LIN {X 0,Y 523.889,Z 260.036,A -85,B 0,C 180,E1 -4743.726,E2 -4743.726} C_VEL
LIN {X 0,Y 523.918,Z 260.038,A -85,B 0,C 180,E1 -4746.691,E2 -4746.691} C_VEL
LIN {X 0,Y 523.956,Z 260.157,A -85,B 0,C 180,E1 -4746.98,E2 -4746.98} C_VEL
LIN {X 0,Y 524.86,Z 266.458,A -85,B 0,C 180,E1 -4748.189,E2 -4748.189} C_VEL
LIN {X 0,Y 524.6,Z 281.046,A -85,B 0,C 180,E1 -4750.841,E2 -4750.841} C_VEL
LIN {X 0,Y 524.215,Z 299.07,A -85,B 0,C 180,E1 -4754.049,E2 -4754.049} C_VEL
LIN {X 0,Y 523.903,Z 316.991,A -85,B 0,C 180,E1 -4757.214,E2 -4757.214} C_VEL
LIN {X 0,Y 523.859,Z 321.977,A -85,B 0,C 180,E1 -4758.092,E2 -4758.092} C_VEL
LIN {X 0,Y 524.896,Z 332.327,A -85,B 0,C 180,E1 -4758.281,E2 -4758.281} C_VEL
LIN {X 0,Y 524.698,Z 397.178,A -85,B 0,C 180,E1 -4759.193,E2 -4759.193} C_VEL
LIN {X 0,Y 524.555,Z 406.795,A -85,B 0,C 180,E1 -4759.41,E2 -4759.41} C_VEL
LIN {X 0,Y 524.415,Z 416.072,A -85,B 0,C 180,E1 -4759.724,E2 -4759.724} C_VEL
LIN {X 0,Y 524.265,Z 425.523,A -85,B 0,C 180,E1 -4760.16,E2 -4760.16} C_VEL
LIN {X 0,Y 524.126,Z 435.206,A -85,B 0,C 180,E1 -4760.742,E2 -4760.742} C_VEL
LIN {X 0,Y 523.895,Z 445.114,A -85,B 0,C 180,E1 -4761.516,E2 -4761.516} C_VEL
LIN {X 0,Y 523.735,Z 452.925,A -85,B 0,C 180,E1 -4762.29,E2 -4762.29} C_VEL
LIN {X 0,Y 523.66,Z 459.358,A -85,B 0,C 180,E1 -4763.064,E2 -4763.064} C_VEL
LIN {X 0,Y 523.588,Z 464.701,A -85,B 0,C 180,E1 -4763.837,E2 -4763.837} C_VEL
LIN {X 0,Y 523.484,Z 469.154,A -85,B 0,C 180,E1 -4764.609,E2 -4764.609} C_VEL
LIN {X 0,Y 523.449,Z 474.389,A -85,B 0,C 180,E1 -4765.767,E2 -4765.767} C_VEL
LIN {X 0,Y 523.406,Z 477.073,A -85,B 0,C 180,E1 -4766.537,E2 -4766.537} C_VEL
LIN {X 0,Y 523.337,Z 480.007,A -85,B 0,C 180,E1 -4767.692,E2 -4767.692} C_VEL
LIN {X 0,Y 523.274,Z 481.275,A -85,B 0,C 180,E1 -4768.462,E2 -4768.462} C_VEL
LIN {X 0,Y 523.25,Z 482.063,A -85,B 0,C 180,E1 -4769.232,E2 -4769.232} C_VEL
LIN {X 0,Y 523.251,Z 482.356,A -85,B 0,C 180,E1 -4770.001,E2 -4770.001} C_VEL
LIN {X 0,Y 523.25,Z 482.054,A -85,B 0,C 180,E1 -4770.771,E2 -4770.771} C_VEL
LIN {X 0,Y 523.274,Z 481.262,A -85,B 0,C 180,E1 -4771.541,E2 -4771.541} C_VEL
LIN {X 0,Y 523.338,Z 479.983,A -85,B 0,C 180,E1 -4772.31,E2 -4772.31} C_VEL
LIN {X 0,Y 523.407,Z 477.038,A -85,B 0,C 180,E1 -4773.465,E2 -4773.465} C_VEL
LIN {X 0,Y 523.45,Z 474.338,A -85,B 0,C 180,E1 -4774.236,E2 -4774.236} C_VEL
LIN {X 0,Y 523.484,Z 469.071,A -85,B 0,C 180,E1 -4775.394,E2 -4775.394} C_VEL
LIN {X 0,Y 523.576,Z 463.108,A -85,B 0,C 180,E1 -4776.405,E2 -4776.405} C_VEL
LIN {X 0,Y 523.705,Z 456.205,A -85,B 0,C 180,E1 -4777.326,E2 -4777.326} C_VEL
LIN {X 0,Y 523.843,Z 448.009,A -85,B 0,C 180,E1 -4778.196,E2 -4778.196} C_VEL
LIN {X 0,Y 523.981,Z 440.157,A -85,B 0,C 180,E1 -4778.874,E2 -4778.874} C_VEL
LIN {X 0,Y 524.132,Z 431.877,A -85,B 0,C 180,E1 -4779.455,E2 -4779.455} C_VEL
LIN {X 0,Y 524.28,Z 421.359,A -85,B 0,C 180,E1 -4780.037,E2 -4780.037} C_VEL
LIN {X 0,Y 524.467,Z 409.445,A -85,B 0,C 180,E1 -4780.497,E2 -4780.497} C_VEL
LIN {X 0,Y 524.616,Z 400.044,A -85,B 0,C 180,E1 -4780.738,E2 -4780.738} C_VEL
LIN {X 0,Y 524.793,Z 362.647,A -85,B 0,C 180,E1 -4781.296,E2 -4781.296} C_VEL
LIN {X 0,Y 524.773,Z 329.873,A -85,B 0,C 180,E1 -4781.752,E2 -4781.752} C_VEL
LIN {X 0,Y 523.817,Z 321.168,A -85,B 0,C 180,E1 -4781.929,E2 -4781.929} C_VEL
LIN {X 0,Y 523.987,Z 304.449,A -85,B 0,C 180,E1 -4784.765,E2 -4784.765} C_VEL
LIN {X 0,Y 524.149,Z 285.845,A -85,B 0,C 180,E1 -4787.822,E2 -4787.822} C_VEL
LIN {X 0,Y 524.255,Z 270.152,A -85,B 0,C 180,E1 -4790.4,E2 -4790.4} C_VEL
LIN {X 0,Y 524.132,Z 261.261,A -85,B 0,C 180,E1 -4791.846,E2 -4791.846} C_VEL
LIN {X 0,Y 523.953,Z 260.033,A -85,B 0,C 180,E1 -4792.061,E2 -4792.061} C_VEL
LIN {X 0,Y 523.897,Z 260.041,A -85,B 0,C 180,E1 -4794.575,E2 -4794.575} C_VEL
LIN {X 0,Y 523.92,Z 260.034,A -85,B 0,C 180,E1 -4797.704,E2 -4797.704} C_VEL
LIN {X 0,Y 523.901,Z 260.042,A -85,B 0,C 180,E1 -4800.845,E2 -4800.845} C_VEL
LIN {X 0,Y 523.863,Z 260.039,A -85,B 0,C 180,E1 -4803.717,E2 -4803.717} C_VEL
LIN {X 0,Y 523.858,Z 260.041,A -85,B 0,C 180,E1 -4806.392,E2 -4806.392} C_VEL
LIN {X 0,Y 523.903,Z 260.04,A -85,B 0,C 180,E1 -4809.087,E2 -4809.087} C_VEL
LIN {X 0,Y 523.898,Z 260.033,A -85,B 0,C 180,E1 -4812.125,E2 -4812.125} C_VEL
LIN {X 0,Y 523.944,Z 260.032,A -85,B 0,C 180,E1 -4815.311,E2 -4815.311} C_VEL
LIN {X 0,Y 523.927,Z 260.034,A -85,B 0,C 180,E1 -4818.694,E2 -4818.694} C_VEL
LIN {X 0,Y 523.922,Z 260.029,A -85,B 0,C 180,E1 -4821.896,E2 -4821.896} C_VEL
LIN {X 0,Y 523.929,Z 260.036,A -85,B 0,C 180,E1 -4824.912,E2 -4824.912} C_VEL
LIN {X 0,Y 523.949,Z 260.029,A -85,B 0,C 180,E1 -4827.679,E2 -4827.679} C_VEL
LIN {X 0,Y 523.966,Z 260.03,A -85,B 0,C 180,E1 -4830.676,E2 -4830.676} C_VEL
LIN {X 0,Y 523.941,Z 260.032,A -85,B 0,C 180,E1 -4833.724,E2 -4833.724} C_VEL
LIN {X 0,Y 523.924,Z 260.033,A -85,B 0,C 180,E1 -4836.267,E2 -4836.267} C_VEL
LIN {X 0,Y 523.958,Z 260.032,A -85,B 0,C 180,E1 -4838.764,E2 -4838.764} C_VEL
LIN {X 0,Y 523.961,Z 260.035,A -85,B 0,C 180,E1 -4841.218,E2 -4841.218} C_VEL
LIN {X 0,Y 524.175,Z 260.008,A -85,B 0,C 180,E1 -4843.643,E2 -4843.643} C_VEL
LIN {X 0,Y 524.071,Z 260.146,A -85,B 0,C 180,E1 -4844.522,E2 -4844.522} C_VEL
LIN {X 0,Y 523.648,Z 275.738,A -85,B 0,C 180,E1 -4846.808,E2 -4846.808} C_VEL
LIN {X 0,Y 523.664,Z 284.072,A -85,B 0,C 180,E1 -4848.14,E2 -4848.14} C_VEL
LIN {X 0,Y 524.911,Z 295.01,A -85,B 0,C 180,E1 -4848.33,E2 -4848.33} C_VEL
LIN {X 0,Y 524.622,Z 361.976,A -85,B 0,C 180,E1 -4849.309,E2 -4849.309} C_VEL
LIN {X 0,Y 524.525,Z 373.079,A -85,B 0,C 180,E1 -4849.6,E2 -4849.6} C_VEL
LIN {X 0,Y 524.355,Z 384.293,A -85,B 0,C 180,E1 -4850.06,E2 -4850.06} C_VEL
LIN {X 0,Y 524.207,Z 393.074,A -85,B 0,C 180,E1 -4850.544,E2 -4850.544} C_VEL
LIN {X 0,Y 524.091,Z 401.438,A -85,B 0,C 180,E1 -4851.125,E2 -4851.125} C_VEL
LIN {X 0,Y 523.938,Z 409.332,A -85,B 0,C 180,E1 -4851.803,E2 -4851.803} C_VEL
LIN {X 0,Y 523.824,Z 415.845,A -85,B 0,C 180,E1 -4852.48,E2 -4852.48} C_VEL
LIN {X 0,Y 523.672,Z 422.247,A -85,B 0,C 180,E1 -4853.281,E2 -4853.281} C_VEL
LIN {X 0,Y 523.616,Z 428.331,A -85,B 0,C 180,E1 -4854.219,E2 -4854.219} C_VEL
LIN {X 0,Y 523.471,Z 434.175,A -85,B 0,C 180,E1 -4855.376,E2 -4855.376} C_VEL
LIN {X 0,Y 523.486,Z 438.418,A -85,B 0,C 180,E1 -4856.533,E2 -4856.533} C_VEL
LIN {X 0,Y 523.339,Z 441.373,A -85,B 0,C 180,E1 -4857.687,E2 -4857.687} C_VEL
LIN {X 0,Y 523.276,Z 442.68,A -85,B 0,C 180,E1 -4858.457,E2 -4858.457} C_VEL
LIN {X 0,Y 523.255,Z 443.496,A -85,B 0,C 180,E1 -4859.227,E2 -4859.227} C_VEL
LIN {X 0,Y 523.256,Z 443.782,A -85,B 0,C 180,E1 -4859.996,E2 -4859.996} C_VEL
LIN {X 0,Y 523.256,Z 443.525,A -85,B 0,C 180,E1 -4860.766,E2 -4860.766} C_VEL
LIN {X 0,Y 523.275,Z 442.784,A -85,B 0,C 180,E1 -4861.535,E2 -4861.535} C_VEL
LIN {X 0,Y 523.34,Z 441.553,A -85,B 0,C 180,E1 -4862.305,E2 -4862.305} C_VEL
LIN {X 0,Y 523.484,Z 438.672,A -85,B 0,C 180,E1 -4863.46,E2 -4863.46} C_VEL
LIN {X 0,Y 523.455,Z 434.53,A -85,B 0,C 180,E1 -4864.616,E2 -4864.616} C_VEL
LIN {X 0,Y 523.613,Z 428.855,A -85,B 0,C 180,E1 -4865.773,E2 -4865.773} C_VEL
LIN {X 0,Y 523.666,Z 422.901,A -85,B 0,C 180,E1 -4866.713,E2 -4866.713} C_VEL
LIN {X 0,Y 523.779,Z 416.652,A -85,B 0,C 180,E1 -4867.513,E2 -4867.513} C_VEL
LIN {X 0,Y 523.983,Z 408.265,A -85,B 0,C 180,E1 -4868.383,E2 -4868.383} C_VEL
LIN {X 0,Y 524.21,Z 398.911,A -85,B 0,C 180,E1 -4869.156,E2 -4869.156} C_VEL
LIN {X 0,Y 524.363,Z 388.078,A -85,B 0,C 180,E1 -4869.835,E2 -4869.835} C_VEL
LIN {X 0,Y 524.504,Z 378.879,A -85,B 0,C 180,E1 -4870.271,E2 -4870.271} C_VEL
LIN {X 0,Y 524.587,Z 369.996,A -85,B 0,C 180,E1 -4870.586,E2 -4870.586} C_VEL
LIN {X 0,Y 524.691,Z 361.16,A -85,B 0,C 180,E1 -4870.804,E2 -4870.804} C_VEL
LIN {X 0,Y 524.859,Z 292.641,A -85,B 0,C 180,E1 -4871.798,E2 -4871.798} C_VEL
LIN {X 0,Y 523.743,Z 285.466,A -85,B 0,C 180,E1 -4871.934,E2 -4871.934} C_VEL
LIN {X 0,Y 523.895,Z 272.16,A -85,B 0,C 180,E1 -4875.01,E2 -4875.01} C_VEL
LIN {X 0,Y 524.015,Z 260.204,A -85,B 0,C 180,E1 -4877.818,E2 -4877.818} C_VEL
LIN {X 0,Y 523.939,Z 260.031,A -85,B 0,C 180,E1 -4880.406,E2 -4880.406} C_VEL
LIN {X 0,Y 523.891,Z 260.042,A -85,B 0,C 180,E1 -4882.889,E2 -4882.889} C_VEL
LIN {X 0,Y 523.88,Z 260.042,A -85,B 0,C 180,E1 -4885.417,E2 -4885.417} C_VEL
LIN {X 0,Y 523.886,Z 260.036,A -85,B 0,C 180,E1 -4887.998,E2 -4887.998} C_VEL
LIN {X 0,Y 523.884,Z 260.039,A -85,B 0,C 180,E1 -4890.87,E2 -4890.87} C_VEL
LIN {X 0,Y 523.934,Z 260.034,A -85,B 0,C 180,E1 -4893.729,E2 -4893.729} C_VEL
LIN {X 0,Y 523.906,Z 260.034,A -85,B 0,C 180,E1 -4894.216,E2 -4894.216} C_VEL
LIN {X 0,Y 523.227,Z 260.121,A -85,B 0,C 180,E1 -4894.857,E2 -4894.857} C_VEL
LIN {X 0,Y 520.334,Z 260.481,A -85,B 0,C 180,E1 -4895.897,E2 -4895.897} C_VEL
LIN {X 0,Y 517.909,Z 260.781,A -85,B 0,C 180,E1 -4896.735,E2 -4896.735} C_VEL
LIN {X 0,Y 516.892,Z 260.913,A -85,B 0,C 180,E1 -4897.383,E2 -4897.383} C_VEL
LIN {X 0,Y 516.822,Z 260.92,A -85,B 0,C 180,E1 -4897.602,E2 -4897.602} C_VEL
LIN {X 0,Y 516.849,Z 260.913,A -85,B 0,C 180,E1 -4900.405,E2 -4900.405} C_VEL
LIN {X 0,Y 516.825,Z 260.916,A -85,B 0,C 180,E1 -4902.829,E2 -4902.829} C_VEL
LIN {X 0,Y 516.86,Z 260.912,A -85,B 0,C 180,E1 -4905.002,E2 -4905.002} C_VEL
LIN {X 0,Y 516.878,Z 260.91,A -85,B 0,C 180,E1 -4908.394,E2 -4908.394} C_VEL
LIN {X 0,Y 516.839,Z 260.916,A -85,B 0,C 180,E1 -4911.279,E2 -4911.279} C_VEL
LIN {X 0,Y 516.845,Z 260.918,A -85,B 0,C 180,E1 -4914.217,E2 -4914.217} C_VEL
LIN {X 0,Y 516.85,Z 260.912,A -85,B 0,C 180,E1 -4917.049,E2 -4917.049} C_VEL
LIN {X 0,Y 516.852,Z 260.918,A -85,B 0,C 180,E1 -4919.793,E2 -4919.793} C_VEL
LIN {X 0,Y 516.88,Z 260.914,A -85,B 0,C 180,E1 -4922.464,E2 -4922.464} C_VEL
LIN {X 0,Y 516.865,Z 260.911,A -85,B 0,C 180,E1 -4925.068,E2 -4925.068} C_VEL
LIN {X 0,Y 516.832,Z 260.921,A -85,B 0,C 180,E1 -4928.459,E2 -4928.459} C_VEL
LIN {X 0,Y 516.849,Z 260.914,A -85,B 0,C 180,E1 -4930.952,E2 -4930.952} C_VEL
LIN {X 0,Y 516.857,Z 260.912,A -85,B 0,C 180,E1 -4933.407,E2 -4933.407} C_VEL
LIN {X 0,Y 516.839,Z 260.915,A -85,B 0,C 180,E1 -4935.831,E2 -4935.831} C_VEL
LIN {X 0,Y 516.946,Z 260.905,A -85,B 0,C 180,E1 -4938.232,E2 -4938.232} C_VEL
LIN {X 0,Y 516.916,Z 260.905,A -85,B 0,C 180,E1 -4941.398,E2 -4941.398} C_VEL
LIN {X 0,Y 517.005,Z 260.9,A -85,B 0,C 180,E1 -4944.538,E2 -4944.538} C_VEL
LIN {X 0,Y 517.022,Z 260.891,A -85,B 0,C 180,E1 -4947.662,E2 -4947.662} C_VEL
LIN {X 0,Y 517.039,Z 260.895,A -85,B 0,C 180,E1 -4950.778,E2 -4950.778} C_VEL
LIN {X 0,Y 516.988,Z 260.901,A -85,B 0,C 180,E1 -4953.116,E2 -4953.116} C_VEL
LIN {X 0,Y 516.949,Z 260.9,A -85,B 0,C 180,E1 -4956.242,E2 -4956.242} C_VEL
LIN {X 0,Y 516.905,Z 260.911,A -85,B 0,C 180,E1 -4959.389,E2 -4959.389} C_VEL
LIN {X 0,Y 516.92,Z 260.905,A -85,B 0,C 180,E1 -4961.824,E2 -4961.824} C_VEL
LIN {X 0,Y 516.88,Z 260.915,A -85,B 0,C 180,E1 -4965.147,E2 -4965.147} C_VEL
LIN {X 0,Y 516.864,Z 260.911,A -85,B 0,C 180,E1 -4968.223,E2 -4968.223} C_VEL
LIN {X 0,Y 516.853,Z 260.913,A -85,B 0,C 180,E1 -4970.702,E2 -4970.702} C_VEL
LIN {X 0,Y 516.817,Z 260.922,A -85,B 0,C 180,E1 -4973.224,E2 -4973.224} C_VEL
LIN {X 0,Y 516.889,Z 260.909,A -85,B 0,C 180,E1 -4976.199,E2 -4976.199} C_VEL
LIN {X 0,Y 516.876,Z 260.913,A -85,B 0,C 180,E1 -4979.305,E2 -4979.305} C_VEL
LIN {X 0,Y 516.843,Z 260.914,A -85,B 0,C 180,E1 -4982.546,E2 -4982.546} C_VEL
LIN {X 0,Y 516.827,Z 260.918,A -85,B 0,C 180,E1 -4985.335,E2 -4985.335} C_VEL
LIN {X 0,Y 516.828,Z 260.921,A -85,B 0,C 180,E1 -4987.946,E2 -4987.946} C_VEL
LIN {X 0,Y 516.866,Z 260.911,A -85,B 0,C 180,E1 -4990.741,E2 -4990.741} C_VEL
LIN {X 0,Y 516.831,Z 260.922,A -85,B 0,C 180,E1 -4993.906,E2 -4993.906} C_VEL
LIN {X 0,Y 516.832,Z 260.921,A -85,B 0,C 180,E1 -4996.11,E2 -4996.11} C_VEL
LIN {X 0,Y 516.856,Z 260.912,A -85,B 0,C 180,E1 -4999.264,E2 -4999.264} C_VEL
LIN {X 0,Y 516.819,Z 260.923,A -85,B 0,C 180,E1 -5002.278,E2 -5002.278} C_VEL
LIN {X 0,Y 516.853,Z 260.913,A -85,B 0,C 180,E1 -5005.18,E2 -5005.18} C_VEL
LIN {X 0,Y 516.835,Z 260.917,A -85,B 0,C 180,E1 -5007.979,E2 -5007.979} C_VEL
LIN {X 0,Y 516.88,Z 260.915,A -85,B 0,C 180,E1 -5010.699,E2 -5010.699} C_VEL
LIN {X 0,Y 516.875,Z 260.91,A -85,B 0,C 180,E1 -5013.815,E2 -5013.815} C_VEL
LIN {X 0,Y 516.823,Z 260.922,A -85,B 0,C 180,E1 -5016.78,E2 -5016.78} C_VEL
LIN {X 0,Y 516.904,Z 260.906,A -85,B 0,C 180,E1 -5019.737,E2 -5019.737} C_VEL
LIN {X 0,Y 516.867,Z 260.916,A -85,B 0,C 180,E1 -5022.599,E2 -5022.599} C_VEL
LIN {X 0,Y 516.911,Z 260.911,A -85,B 0,C 180,E1 -5025.034,E2 -5025.034} C_VEL
LIN {X 0,Y 516.94,Z 260.902,A -85,B 0,C 180,E1 -5028.238,E2 -5028.238} C_VEL
LIN {X 0,Y 516.927,Z 260.908,A -85,B 0,C 180,E1 -5031.403,E2 -5031.403} C_VEL
LIN {X 0,Y 516.962,Z 260.9,A -85,B 0,C 180,E1 -5033.761,E2 -5033.761} C_VEL
LIN {X 0,Y 516.954,Z 260.904,A -85,B 0,C 180,E1 -5036.887,E2 -5036.887} C_VEL
LIN {X 0,Y 517.075,Z 260.891,A -85,B 0,C 180,E1 -5039.225,E2 -5039.225} C_VEL
LIN {X 0,Y 517.056,Z 260.887,A -85,B 0,C 180,E1 -5042.341,E2 -5042.341} C_VEL
LIN {X 0,Y 516.995,Z 260.901,A -85,B 0,C 180,E1 -5045.464,E2 -5045.464} C_VEL
LIN {X 0,Y 516.938,Z 260.901,A -85,B 0,C 180,E1 -5048.604,E2 -5048.604} C_VEL
LIN {X 0,Y 516.94,Z 260.907,A -85,B 0,C 180,E1 -5051.81,E2 -5051.81} C_VEL
LIN {X 0,Y 516.932,Z 260.904,A -85,B 0,C 180,E1 -5055.149,E2 -5055.149} C_VEL
LIN {X 0,Y 516.867,Z 260.914,A -85,B 0,C 180,E1 -5058.227,E2 -5058.227} C_VEL
LIN {X 0,Y 516.89,Z 260.908,A -85,B 0,C 180,E1 -5060.705,E2 -5060.705} C_VEL
LIN {X 0,Y 516.848,Z 260.913,A -85,B 0,C 180,E1 -5063.227,E2 -5063.227} C_VEL
LIN {X 0,Y 516.872,Z 260.915,A -85,B 0,C 180,E1 -5066.185,E2 -5066.185} C_VEL
LIN {X 0,Y 516.914,Z 260.905,A -85,B 0,C 180,E1 -5069.308,E2 -5069.308} C_VEL
LIN {X 0,Y 516.888,Z 260.912,A -85,B 0,C 180,E1 -5072.546,E2 -5072.546} C_VEL
LIN {X 0,Y 516.848,Z 260.913,A -85,B 0,C 180,E1 -5075.33,E2 -5075.33} C_VEL
LIN {X 0,Y 516.866,Z 260.915,A -85,B 0,C 180,E1 -5078.72,E2 -5078.72} C_VEL
LIN {X 0,Y 516.849,Z 260.914,A -85,B 0,C 180,E1 -5081.784,E2 -5081.784} C_VEL
LIN {X 0,Y 516.893,Z 260.91,A -85,B 0,C 180,E1 -5085.009,E2 -5085.009} C_VEL
LIN {X 0,Y 516.852,Z 260.918,A -85,B 0,C 180,E1 -5088.409,E2 -5088.409} C_VEL
LIN {X 0,Y 516.873,Z 260.911,A -85,B 0,C 180,E1 -5091.286,E2 -5091.286} C_VEL
LIN {X 0,Y 516.854,Z 260.914,A -85,B 0,C 180,E1 -5094.221,E2 -5094.221} C_VEL
LIN {X 0,Y 516.878,Z 260.915,A -85,B 0,C 180,E1 -5097.054,E2 -5097.054} C_VEL
LIN {X 0,Y 516.85,Z 260.913,A -85,B 0,C 180,E1 -5099.796,E2 -5099.796} C_VEL
LIN {X 0,Y 516.868,Z 260.912,A -85,B 0,C 180,E1 -5102.466,E2 -5102.466} C_VEL
LIN {X 0,Y 516.87,Z 260.915,A -85,B 0,C 180,E1 -5105.648,E2 -5105.648} C_VEL
LIN {X 0,Y 516.903,Z 260.981,A -85,B 0,C 180,E1 -5106.832,E2 -5106.832} C_VEL
LIN {X 0,Y 517.891,Z 267.442,A -85,B 0,C 180,E1 -5108.089,E2 -5108.089} C_VEL
LIN {X 0,Y 517.585,Z 281.977,A -85,B 0,C 180,E1 -5110.777,E2 -5110.777} C_VEL
LIN {X 0,Y 517.177,Z 298.875,A -85,B 0,C 180,E1 -5113.826,E2 -5113.826} C_VEL
LIN {X 0,Y 516.885,Z 315.646,A -85,B 0,C 180,E1 -5116.837,E2 -5116.837} C_VEL
LIN {X 0,Y 516.816,Z 321.814,A -85,B 0,C 180,E1 -5117.939,E2 -5117.939} C_VEL
LIN {X 0,Y 517.959,Z 331.933,A -85,B 0,C 180,E1 -5118.121,E2 -5118.121} C_VEL
LIN {X 0,Y 517.695,Z 397.549,A -85,B 0,C 180,E1 -5119.07,E2 -5119.07} C_VEL
LIN {X 0,Y 517.537,Z 407.745,A -85,B 0,C 180,E1 -5119.314,E2 -5119.314} C_VEL
LIN {X 0,Y 517.367,Z 417.888,A -85,B 0,C 180,E1 -5119.682,E2 -5119.682} C_VEL
LIN {X 0,Y 517.166,Z 428.671,A -85,B 0,C 180,E1 -5120.221,E2 -5120.221} C_VEL
LIN {X 0,Y 516.991,Z 438.738,A -85,B 0,C 180,E1 -5120.909,E2 -5120.909} C_VEL
LIN {X 0,Y 516.813,Z 446.774,A -85,B 0,C 180,E1 -5121.595,E2 -5121.595} C_VEL
LIN {X 0,Y 516.692,Z 452.559,A -85,B 0,C 180,E1 -5122.184,E2 -5122.184} C_VEL
LIN {X 0,Y 516.593,Z 459.014,A -85,B 0,C 180,E1 -5122.968,E2 -5122.968} C_VEL
LIN {X 0,Y 516.495,Z 464.377,A -85,B 0,C 180,E1 -5123.752,E2 -5123.752} C_VEL
LIN {X 0,Y 516.421,Z 468.849,A -85,B 0,C 180,E1 -5124.535,E2 -5124.535} C_VEL
LIN {X 0,Y 516.34,Z 474.1,A -85,B 0,C 180,E1 -5125.708,E2 -5125.708} C_VEL
LIN {X 0,Y 516.324,Z 476.795,A -85,B 0,C 180,E1 -5126.49,E2 -5126.49} C_VEL
LIN {X 0,Y 516.264,Z 479.741,A -85,B 0,C 180,E1 -5127.661,E2 -5127.661} C_VEL
LIN {X 0,Y 516.192,Z 481.013,A -85,B 0,C 180,E1 -5128.441,E2 -5128.441} C_VEL
LIN {X 0,Y 516.16,Z 481.804,A -85,B 0,C 180,E1 -5129.221,E2 -5129.221} C_VEL
LIN {X 0,Y 516.158,Z 482.095,A -85,B 0,C 180,E1 -5130.001,E2 -5130.001} C_VEL
LIN {X 0,Y 516.16,Z 481.79,A -85,B 0,C 180,E1 -5130.781,E2 -5130.781} C_VEL
LIN {X 0,Y 516.192,Z 480.994,A -85,B 0,C 180,E1 -5131.562,E2 -5131.562} C_VEL
LIN {X 0,Y 516.264,Z 479.708,A -85,B 0,C 180,E1 -5132.342,E2 -5132.342} C_VEL
LIN {X 0,Y 516.325,Z 476.742,A -85,B 0,C 180,E1 -5133.513,E2 -5133.513} C_VEL
LIN {X 0,Y 516.341,Z 474.032,A -85,B 0,C 180,E1 -5134.295,E2 -5134.295} C_VEL
LIN {X 0,Y 516.422,Z 468.734,A -85,B 0,C 180,E1 -5135.468,E2 -5135.468} C_VEL
LIN {X 0,Y 516.508,Z 461.774,A -85,B 0,C 180,E1 -5136.634,E2 -5136.634} C_VEL
LIN {X 0,Y 516.628,Z 455.794,A -85,B 0,C 180,E1 -5137.427,E2 -5137.427} C_VEL
LIN {X 0,Y 516.761,Z 447.559,A -85,B 0,C 180,E1 -5138.31,E2 -5138.31} C_VEL
LIN {X 0,Y 516.945,Z 439.657,A -85,B 0,C 180,E1 -5138.996,E2 -5138.996} C_VEL
LIN {X 0,Y 517.083,Z 431.321,A -85,B 0,C 180,E1 -5139.585,E2 -5139.585} C_VEL
LIN {X 0,Y 517.284,Z 420.731,A -85,B 0,C 180,E1 -5140.174,E2 -5140.174} C_VEL
LIN {X 0,Y 517.463,Z 409.407,A -85,B 0,C 180,E1 -5140.616,E2 -5140.616} C_VEL
LIN {X 0,Y 517.618,Z 400.166,A -85,B 0,C 180,E1 -5140.86,E2 -5140.86} C_VEL
LIN {X 0,Y 517.778,Z 370.892,A -85,B 0,C 180,E1 -5141.313,E2 -5141.313} C_VEL
LIN {X 0,Y 517.811,Z 330.227,A -85,B 0,C 180,E1 -5141.902,E2 -5141.902} C_VEL
LIN {X 0,Y 516.737,Z 320.994,A -85,B 0,C 180,E1 -5142.071,E2 -5142.071} C_VEL
LIN {X 0,Y 516.909,Z 302.864,A -85,B 0,C 180,E1 -5145.128,E2 -5145.128} C_VEL
LIN {X 0,Y 517.047,Z 287.661,A -85,B 0,C 180,E1 -5147.669,E2 -5147.669} C_VEL
LIN {X 0,Y 517.201,Z 272.926,A -85,B 0,C 180,E1 -5150.104,E2 -5150.104} C_VEL
LIN {X 0,Y 517.192,Z 262.999,A -85,B 0,C 180,E1 -5151.735,E2 -5151.735} C_VEL
LIN {X 0,Y 516.906,Z 260.911,A -85,B 0,C 180,E1 -5152.115,E2 -5152.115} C_VEL
LIN {X 0,Y 516.833,Z 260.923,A -85,B 0,C 180,E1 -5154.933,E2 -5154.933} C_VEL
LIN {X 0,Y 516.864,Z 260.913,A -85,B 0,C 180,E1 -5157.89,E2 -5157.89} C_VEL
LIN {X 0,Y 516.854,Z 260.918,A -85,B 0,C 180,E1 -5161.113,E2 -5161.113} C_VEL
LIN {X 0,Y 516.829,Z 260.915,A -85,B 0,C 180,E1 -5163.951,E2 -5163.951} C_VEL
LIN {X 0,Y 516.803,Z 260.924,A -85,B 0,C 180,E1 -5166.753,E2 -5166.753} C_VEL
LIN {X 0,Y 516.838,Z 260.913,A -85,B 0,C 180,E1 -5169.726,E2 -5169.726} C_VEL
LIN {X 0,Y 516.849,Z 260.919,A -85,B 0,C 180,E1 -5172.836,E2 -5172.836} C_VEL
LIN {X 0,Y 516.91,Z 260.912,A -85,B 0,C 180,E1 -5175.006,E2 -5175.006} C_VEL
LIN {X 0,Y 516.863,Z 260.91,A -85,B 0,C 180,E1 -5178.406,E2 -5178.406} C_VEL
LIN {X 0,Y 516.886,Z 260.911,A -85,B 0,C 180,E1 -5181.282,E2 -5181.282} C_VEL
LIN {X 0,Y 516.87,Z 260.909,A -85,B 0,C 180,E1 -5184.217,E2 -5184.217} C_VEL
LIN {X 0,Y 516.895,Z 260.914,A -85,B 0,C 180,E1 -5187.05,E2 -5187.05} C_VEL
LIN {X 0,Y 516.884,Z 260.909,A -85,B 0,C 180,E1 -5189.793,E2 -5189.793} C_VEL
LIN {X 0,Y 516.893,Z 260.909,A -85,B 0,C 180,E1 -5192.463,E2 -5192.463} C_VEL
LIN {X 0,Y 516.873,Z 260.919,A -85,B 0,C 180,E1 -5195.067,E2 -5195.067} C_VEL
LIN {X 0,Y 516.883,Z 260.913,A -85,B 0,C 180,E1 -5197.619,E2 -5197.619} C_VEL
LIN {X 0,Y 516.944,Z 260.901,A -85,B 0,C 180,E1 -5200.127,E2 -5200.127} C_VEL
LIN {X 0,Y 517.085,Z 260.892,A -85,B 0,C 180,E1 -5203.413,E2 -5203.413} C_VEL
LIN {X 0,Y 516.978,Z 261.072,A -85,B 0,C 180,E1 -5204.565,E2 -5204.565} C_VEL
LIN {X 0,Y 516.589,Z 276.65,A -85,B 0,C 180,E1 -5206.825,E2 -5206.825} C_VEL
LIN {X 0,Y 516.632,Z 284.166,A -85,B 0,C 180,E1 -5207.976,E2 -5207.976} C_VEL
LIN {X 0,Y 517.975,Z 295.466,A -85,B 0,C 180,E1 -5208.178,E2 -5208.178} C_VEL
LIN {X 0,Y 517.648,Z 362.688,A -85,B 0,C 180,E1 -5209.188,E2 -5209.188} C_VEL
LIN {X 0,Y 517.533,Z 373.605,A -85,B 0,C 180,E1 -5209.482,E2 -5209.482} C_VEL
LIN {X 0,Y 517.354,Z 384.247,A -85,B 0,C 180,E1 -5209.924,E2 -5209.924} C_VEL
LIN {X 0,Y 517.2,Z 393.084,A -85,B 0,C 180,E1 -5210.415,E2 -5210.415} C_VEL
LIN {X 0,Y 517.087,Z 401.494,A -85,B 0,C 180,E1 -5211.004,E2 -5211.004} C_VEL
LIN {X 0,Y 516.923,Z 409.433,A -85,B 0,C 180,E1 -5211.691,E2 -5211.691} C_VEL
LIN {X 0,Y 516.782,Z 415.979,A -85,B 0,C 180,E1 -5212.377,E2 -5212.377} C_VEL
LIN {X 0,Y 516.628,Z 421.824,A -85,B 0,C 180,E1 -5213.11,E2 -5213.11} C_VEL
LIN {X 0,Y 516.628,Z 427.34,A -85,B 0,C 180,E1 -5213.945,E2 -5213.945} C_VEL
LIN {X 0,Y 516.399,Z 432.588,A -85,B 0,C 180,E1 -5214.921,E2 -5214.921} C_VEL
LIN {X 0,Y 516.387,Z 437.439,A -85,B 0,C 180,E1 -5216.094,E2 -5216.094} C_VEL
LIN {X 0,Y 516.375,Z 439.806,A -85,B 0,C 180,E1 -5216.875,E2 -5216.875} C_VEL
LIN {X 0,Y 516.269,Z 441.617,A -85,B 0,C 180,E1 -5217.656,E2 -5217.656} C_VEL
LIN {X 0,Y 516.193,Z 442.925,A -85,B 0,C 180,E1 -5218.436,E2 -5218.436} C_VEL
LIN {X 0,Y 516.165,Z 443.747,A -85,B 0,C 180,E1 -5219.216,E2 -5219.216} C_VEL
LIN {X 0,Y 516.163,Z 444.044,A -85,B 0,C 180,E1 -5219.996,E2 -5219.996} C_VEL
LIN {X 0,Y 516.166,Z 443.772,A -85,B 0,C 180,E1 -5220.776,E2 -5220.776} C_VEL
LIN {X 0,Y 516.192,Z 443.021,A -85,B 0,C 180,E1 -5221.556,E2 -5221.556} C_VEL
LIN {X 0,Y 516.269,Z 441.784,A -85,B 0,C 180,E1 -5222.337,E2 -5222.337} C_VEL
LIN {X 0,Y 516.389,Z 438.889,A -85,B 0,C 180,E1 -5223.507,E2 -5223.507} C_VEL
LIN {X 0,Y 516.366,Z 434.728,A -85,B 0,C 180,E1 -5224.68,E2 -5224.68} C_VEL
LIN {X 0,Y 516.57,Z 429.033,A -85,B 0,C 180,E1 -5225.852,E2 -5225.852} C_VEL
LIN {X 0,Y 516.616,Z 423.523,A -85,B 0,C 180,E1 -5226.737,E2 -5226.737} C_VEL
LIN {X 0,Y 516.74,Z 416.759,A -85,B 0,C 180,E1 -5227.616,E2 -5227.616} C_VEL
LIN {X 0,Y 516.918,Z 409.364,A -85,B 0,C 180,E1 -5228.4,E2 -5228.4} C_VEL
LIN {X 0,Y 517.114,Z 401.449,A -85,B 0,C 180,E1 -5229.086,E2 -5229.086} C_VEL
LIN {X 0,Y 517.303,Z 391.56,A -85,B 0,C 180,E1 -5229.773,E2 -5229.773} C_VEL
LIN {X 0,Y 517.487,Z 381.153,A -85,B 0,C 180,E1 -5230.313,E2 -5230.313} C_VEL
LIN {X 0,Y 517.604,Z 370.556,A -85,B 0,C 180,E1 -5230.706,E2 -5230.706} C_VEL
LIN {X 0,Y 517.688,Z 361.917,A -85,B 0,C 180,E1 -5230.927,E2 -5230.927} C_VEL
LIN {X 0,Y 517.821,Z 292.671,A -85,B 0,C 180,E1 -5231.961,E2 -5231.961} C_VEL
LIN {X 0,Y 516.713,Z 285.633,A -85,B 0,C 180,E1 -5232.099,E2 -5232.099} C_VEL
LIN {X 0,Y 516.859,Z 272.721,A -85,B 0,C 180,E1 -5235.109,E2 -5235.109} C_VEL
LIN {X 0,Y 517.04,Z 262.042,A -85,B 0,C 180,E1 -5237.641,E2 -5237.641} C_VEL
LIN {X 0,Y 516.929,Z 260.907,A -85,B 0,C 180,E1 -5237.946,E2 -5237.946} C_VEL
LIN {X 0,Y 516.888,Z 260.912,A -85,B 0,C 180,E1 -5240.697,E2 -5240.697} C_VEL
LIN {X 0,Y 516.841,Z 260.92,A -85,B 0,C 180,E1 -5243.219,E2 -5243.219} C_VEL
LIN {X 0,Y 516.863,Z 260.911,A -85,B 0,C 180,E1 -5246.177,E2 -5246.177} C_VEL
LIN {X 0,Y 516.882,Z 260.914,A -85,B 0,C 180,E1 -5249.301,E2 -5249.301} C_VEL
LIN {X 0,Y 516.87,Z 260.91,A -85,B 0,C 180,E1 -5252.538,E2 -5252.538} C_VEL
LIN {X 0,Y 516.837,Z 260.92,A -85,B 0,C 180,E1 -5255.324,E2 -5255.324} C_VEL
LIN {X 0,Y 516.822,Z 260.92,A -85,B 0,C 180,E1 -5257.602,E2 -5257.602} C_VEL
LIN {X 0,Y 516.188,Z 261.004,A -85,B 0,C 180,E1 -5258.252,E2 -5258.252} C_VEL
LIN {X 0,Y 513.335,Z 261.357,A -85,B 0,C 180,E1 -5259.308,E2 -5259.308} C_VEL
LIN {X 0,Y 510.908,Z 261.654,A -85,B 0,C 180,E1 -5260.158,E2 -5260.158} C_VEL
LIN {X 0,Y 509.874,Z 261.782,A -85,B 0,C 180,E1 -5260.814,E2 -5260.814} C_VEL
LIN {X 0,Y 509.795,Z 261.793,A -85,B 0,C 180,E1 -5261.037,E2 -5261.037} C_VEL
LIN {X 0,Y 509.787,Z 261.795,A -85,B 0,C 180,E1 -5264.202,E2 -5264.202} C_VEL
LIN {X 0,Y 509.786,Z 261.793,A -85,B 0,C 180,E1 -5266.933,E2 -5266.933} C_VEL
LIN {X 0,Y 509.799,Z 261.797,A -85,B 0,C 180,E1 -5269.613,E2 -5269.613} C_VEL
LIN {X 0,Y 509.777,Z 261.794,A -85,B 0,C 180,E1 -5272.655,E2 -5272.655} C_VEL
LIN {X 0,Y 509.815,Z 261.795,A -85,B 0,C 180,E1 -5275.793,E2 -5275.793} C_VEL
LIN {X 0,Y 509.8,Z 261.792,A -85,B 0,C 180,E1 -5278.716,E2 -5278.716} C_VEL
LIN {X 0,Y 509.849,Z 261.791,A -85,B 0,C 180,E1 -5281.895,E2 -5281.895} C_VEL
LIN {X 0,Y 509.831,Z 261.79,A -85,B 0,C 180,E1 -5284.7,E2 -5284.7} C_VEL
LIN {X 0,Y 509.775,Z 261.794,A -85,B 0,C 180,E1 -5287.454,E2 -5287.454} C_VEL
LIN {X 0,Y 509.862,Z 261.786,A -85,B 0,C 180,E1 -5289.841,E2 -5289.841} C_VEL
LIN {X 0,Y 509.828,Z 261.788,A -85,B 0,C 180,E1 -5293.172,E2 -5293.172} C_VEL
LIN {X 0,Y 509.807,Z 261.79,A -85,B 0,C 180,E1 -5295.631,E2 -5295.631} C_VEL
LIN {X 0,Y 509.872,Z 261.787,A -85,B 0,C 180,E1 -5298.872,E2 -5298.872} C_VEL
LIN {X 0,Y 509.893,Z 261.781,A -85,B 0,C 180,E1 -5302.076,E2 -5302.076} C_VEL
LIN {X 0,Y 509.951,Z 261.777,A -85,B 0,C 180,E1 -5304.463,E2 -5304.463} C_VEL
LIN {X 0,Y 509.995,Z 261.767,A -85,B 0,C 180,E1 -5307.629,E2 -5307.629} C_VEL
LIN {X 0,Y 509.99,Z 261.767,A -85,B 0,C 180,E1 -5309.999,E2 -5309.999} C_VEL
LIN {X 0,Y 509.929,Z 261.78,A -85,B 0,C 180,E1 -5313.159,E2 -5313.159} C_VEL
LIN {X 0,Y 509.917,Z 261.777,A -85,B 0,C 180,E1 -5316.329,E2 -5316.329} C_VEL
LIN {X 0,Y 509.889,Z 261.783,A -85,B 0,C 180,E1 -5318.719,E2 -5318.719} C_VEL
LIN {X 0,Y 509.888,Z 261.781,A -85,B 0,C 180,E1 -5321.93,E2 -5321.93} C_VEL
LIN {X 0,Y 509.83,Z 261.793,A -85,B 0,C 180,E1 -5325.242,E2 -5325.242} C_VEL
LIN {X 0,Y 509.826,Z 261.789,A -85,B 0,C 180,E1 -5328.002,E2 -5328.002} C_VEL
LIN {X 0,Y 509.792,Z 261.795,A -85,B 0,C 180,E1 -5331.002,E2 -5331.002} C_VEL
LIN {X 0,Y 509.782,Z 261.799,A -85,B 0,C 180,E1 -5333.564,E2 -5333.564} C_VEL
LIN {X 0,Y 509.857,Z 261.784,A -85,B 0,C 180,E1 -5336.381,E2 -5336.381} C_VEL
LIN {X 0,Y 509.826,Z 261.788,A -85,B 0,C 180,E1 -5338.845,E2 -5338.845} C_VEL
LIN {X 0,Y 509.769,Z 261.801,A -85,B 0,C 180,E1 -5341.592,E2 -5341.592} C_VEL
LIN {X 0,Y 509.798,Z 261.793,A -85,B 0,C 180,E1 -5344.415,E2 -5344.415} C_VEL
LIN {X 0,Y 509.764,Z 261.797,A -85,B 0,C 180,E1 -5347.343,E2 -5347.343} C_VEL
LIN {X 0,Y 509.83,Z 261.791,A -85,B 0,C 180,E1 -5350.381,E2 -5350.381} C_VEL
LIN {X 0,Y 509.789,Z 261.792,A -85,B 0,C 180,E1 -5353.067,E2 -5353.067} C_VEL
LIN {X 0,Y 509.78,Z 261.798,A -85,B 0,C 180,E1 -5355.795,E2 -5355.795} C_VEL
LIN {X 0,Y 509.817,Z 261.793,A -85,B 0,C 180,E1 -5358.579,E2 -5358.579} C_VEL
LIN {X 0,Y 509.806,Z 261.793,A -85,B 0,C 180,E1 -5361.79,E2 -5361.79} C_VEL
LIN {X 0,Y 509.803,Z 261.796,A -85,B 0,C 180,E1 -5364.627,E2 -5364.627} C_VEL
LIN {X 0,Y 509.822,Z 261.788,A -85,B 0,C 180,E1 -5367.485,E2 -5367.485} C_VEL
LIN {X 0,Y 509.818,Z 261.794,A -85,B 0,C 180,E1 -5370.278,E2 -5370.278} C_VEL
LIN {X 0,Y 509.839,Z 261.79,A -85,B 0,C 180,E1 -5372.948,E2 -5372.948} C_VEL
LIN {X 0,Y 509.806,Z 261.79,A -85,B 0,C 180,E1 -5375.577,E2 -5375.577} C_VEL
LIN {X 0,Y 509.787,Z 261.794,A -85,B 0,C 180,E1 -5378.153,E2 -5378.153} C_VEL
LIN {X 0,Y 509.825,Z 261.794,A -85,B 0,C 180,E1 -5380.685,E2 -5380.685} C_VEL
LIN {X 0,Y 509.839,Z 261.791,A -85,B 0,C 180,E1 -5383.178,E2 -5383.178} C_VEL
LIN {X 0,Y 509.828,Z 261.788,A -85,B 0,C 180,E1 -5385.638,E2 -5385.638} C_VEL
LIN {X 0,Y 509.884,Z 261.787,A -85,B 0,C 180,E1 -5388.879,E2 -5388.879} C_VEL
LIN {X 0,Y 509.896,Z 261.779,A -85,B 0,C 180,E1 -5392.082,E2 -5392.082} C_VEL
LIN {X 0,Y 509.946,Z 261.774,A -85,B 0,C 180,E1 -5394.468,E2 -5394.468} C_VEL
LIN {X 0,Y 510.025,Z 261.767,A -85,B 0,C 180,E1 -5397.635,E2 -5397.635} C_VEL
LIN {X 0,Y 510.014,Z 261.765,A -85,B 0,C 180,E1 -5400.004,E2 -5400.004} C_VEL
LIN {X 0,Y 510.027,Z 261.763,A -85,B 0,C 180,E1 -5402.373,E2 -5402.373} C_VEL
LIN {X 0,Y 509.946,Z 261.778,A -85,B 0,C 180,E1 -5405.54,E2 -5405.54} C_VEL
LIN {X 0,Y 509.887,Z 261.78,A -85,B 0,C 180,E1 -5408.724,E2 -5408.724} C_VEL
LIN {X 0,Y 509.892,Z 261.784,A -85,B 0,C 180,E1 -5411.935,E2 -5411.935} C_VEL
LIN {X 0,Y 509.884,Z 261.783,A -85,B 0,C 180,E1 -5415.245,E2 -5415.245} C_VEL
LIN {X 0,Y 509.827,Z 261.789,A -85,B 0,C 180,E1 -5418.488,E2 -5418.488} C_VEL
LIN {X 0,Y 509.833,Z 261.787,A -85,B 0,C 180,E1 -5421.005,E2 -5421.005} C_VEL
LIN {X 0,Y 509.81,Z 261.793,A -85,B 0,C 180,E1 -5423.567,E2 -5423.567} C_VEL
LIN {X 0,Y 509.808,Z 261.794,A -85,B 0,C 180,E1 -5426.36,E2 -5426.36} C_VEL
LIN {X 0,Y 509.843,Z 261.786,A -85,B 0,C 180,E1 -5428.849,E2 -5428.849} C_VEL
LIN {X 0,Y 509.813,Z 261.791,A -85,B 0,C 180,E1 -5431.593,E2 -5431.593} C_VEL
LIN {X 0,Y 509.828,Z 261.793,A -85,B 0,C 180,E1 -5434.418,E2 -5434.418} C_VEL
LIN {X 0,Y 509.787,Z 261.792,A -85,B 0,C 180,E1 -5437.346,E2 -5437.346} C_VEL
LIN {X 0,Y 509.809,Z 261.795,A -85,B 0,C 180,E1 -5440.387,E2 -5440.387} C_VEL
LIN {X 0,Y 509.803,Z 261.79,A -85,B 0,C 180,E1 -5443.576,E2 -5443.576} C_VEL
LIN {X 0,Y 509.79,Z 261.799,A -85,B 0,C 180,E1 -5446.428,E2 -5446.428} C_VEL
LIN {X 0,Y 509.812,Z 261.789,A -85,B 0,C 180,E1 -5449.618,E2 -5449.618} C_VEL
LIN {X 0,Y 509.804,Z 261.797,A -85,B 0,C 180,E1 -5452.66,E2 -5452.66} C_VEL
LIN {X 0,Y 509.837,Z 261.786,A -85,B 0,C 180,E1 -5455.803,E2 -5455.803} C_VEL
LIN {X 0,Y 509.837,Z 261.793,A -85,B 0,C 180,E1 -5458.724,E2 -5458.724} C_VEL
LIN {X 0,Y 509.834,Z 261.792,A -85,B 0,C 180,E1 -5461.155,E2 -5461.155} C_VEL
LIN {X 0,Y 509.836,Z 261.787,A -85,B 0,C 180,E1 -5463.827,E2 -5463.827} C_VEL
LIN {X 0,Y 509.862,Z 261.934,A -85,B 0,C 180,E1 -5466.709,E2 -5466.709} C_VEL
LIN {X 0,Y 510.885,Z 268.395,A -85,B 0,C 180,E1 -5467.986,E2 -5467.986} C_VEL
LIN {X 0,Y 510.636,Z 281.817,A -85,B 0,C 180,E1 -5470.505,E2 -5470.505} C_VEL
LIN {X 0,Y 510.184,Z 298.655,A -85,B 0,C 180,E1 -5473.598,E2 -5473.598} C_VEL
LIN {X 0,Y 509.851,Z 315.417,A -85,B 0,C 180,E1 -5476.652,E2 -5476.652} C_VEL
LIN {X 0,Y 509.744,Z 321.538,A -85,B 0,C 180,E1 -5477.76,E2 -5477.76} C_VEL
LIN {X 0,Y 511.011,Z 333.503,A -85,B 0,C 180,E1 -5477.985,E2 -5477.985} C_VEL
LIN {X 0,Y 510.677,Z 399.137,A -85,B 0,C 180,E1 -5478.968,E2 -5478.968} C_VEL
LIN {X 0,Y 510.491,Z 409.487,A -85,B 0,C 180,E1 -5479.24,E2 -5479.24} C_VEL
LIN {X 0,Y 510.306,Z 420.72,A -85,B 0,C 180,E1 -5479.688,E2 -5479.688} C_VEL
LIN {X 0,Y 510.09,Z 431.258,A -85,B 0,C 180,E1 -5480.285,E2 -5480.285} C_VEL
LIN {X 0,Y 509.92,Z 439.549,A -85,B 0,C 180,E1 -5480.882,E2 -5480.882} C_VEL
LIN {X 0,Y 509.741,Z 447.413,A -85,B 0,C 180,E1 -5481.578,E2 -5481.578} C_VEL
LIN {X 0,Y 509.582,Z 453.913,A -85,B 0,C 180,E1 -5482.274,E2 -5482.274} C_VEL
LIN {X 0,Y 509.492,Z 460.54,A -85,B 0,C 180,E1 -5483.129,E2 -5483.129} C_VEL
LIN {X 0,Y 509.37,Z 467.567,A -85,B 0,C 180,E1 -5484.26,E2 -5484.26} C_VEL
LIN {X 0,Y 509.225,Z 472.277,A -85,B 0,C 180,E1 -5485.251,E2 -5485.251} C_VEL
LIN {X 0,Y 509.258,Z 475.327,A -85,B 0,C 180,E1 -5486.045,E2 -5486.045} C_VEL
LIN {X 0,Y 509.213,Z 477.688,A -85,B 0,C 180,E1 -5486.837,E2 -5486.837} C_VEL
LIN {X 0,Y 509.193,Z 479.475,A -85,B 0,C 180,E1 -5487.628,E2 -5487.628} C_VEL
LIN {X 0,Y 509.113,Z 480.751,A -85,B 0,C 180,E1 -5488.419,E2 -5488.419} C_VEL
LIN {X 0,Y 509.074,Z 481.544,A -85,B 0,C 180,E1 -5489.21,E2 -5489.21} C_VEL
LIN {X 0,Y 509.07,Z 481.835,A -85,B 0,C 180,E1 -5490.001,E2 -5490.001} C_VEL
LIN {X 0,Y 509.074,Z 481.526,A -85,B 0,C 180,E1 -5490.792,E2 -5490.792} C_VEL
LIN {X 0,Y 509.113,Z 480.722,A -85,B 0,C 180,E1 -5491.583,E2 -5491.583} C_VEL
LIN {X 0,Y 509.193,Z 479.433,A -85,B 0,C 180,E1 -5492.374,E2 -5492.374} C_VEL
LIN {X 0,Y 509.245,Z 476.445,A -85,B 0,C 180,E1 -5493.562,E2 -5493.562} C_VEL
LIN {X 0,Y 509.235,Z 473.721,A -85,B 0,C 180,E1 -5494.355,E2 -5494.355} C_VEL
LIN {X 0,Y 509.337,Z 468.397,A -85,B 0,C 180,E1 -5495.544,E2 -5495.544} C_VEL
LIN {X 0,Y 509.463,Z 461.271,A -85,B 0,C 180,E1 -5496.744,E2 -5496.744} C_VEL
LIN {X 0,Y 509.543,Z 455.383,A -85,B 0,C 180,E1 -5497.53,E2 -5497.53} C_VEL
LIN {X 0,Y 509.68,Z 448.139,A -85,B 0,C 180,E1 -5498.326,E2 -5498.326} C_VEL
LIN {X 0,Y 509.866,Z 440.403,A -85,B 0,C 180,E1 -5499.022,E2 -5499.022} C_VEL
LIN {X 0,Y 510.024,Z 432.285,A -85,B 0,C 180,E1 -5499.619,E2 -5499.619} C_VEL
LIN {X 0,Y 510.174,Z 423.89,A -85,B 0,C 180,E1 -5500.117,E2 -5500.117} C_VEL
LIN {X 0,Y 510.415,Z 415.358,A -85,B 0,C 180,E1 -5500.513,E2 -5500.513} C_VEL
LIN {X 0,Y 510.495,Z 406.064,A -85,B 0,C 180,E1 -5500.838,E2 -5500.838} C_VEL
LIN {X 0,Y 510.708,Z 395.239,A -85,B 0,C 180,E1 -5501.084,E2 -5501.084} C_VEL
LIN {X 0,Y 510.854,Z 330.818,A -85,B 0,C 180,E1 -5502.052,E2 -5502.052} C_VEL
LIN {X 0,Y 509.653,Z 320.665,A -85,B 0,C 180,E1 -5502.244,E2 -5502.244} C_VEL
LIN {X 0,Y 509.86,Z 304.561,A -85,B 0,C 180,E1 -5504.979,E2 -5504.979} C_VEL
LIN {X 0,Y 510.039,Z 286.907,A -85,B 0,C 180,E1 -5507.946,E2 -5507.946} C_VEL
LIN {X 0,Y 510.187,Z 270.494,A -85,B 0,C 180,E1 -5510.686,E2 -5510.686} C_VEL
LIN {X 0,Y 510.124,Z 263.557,A -85,B 0,C 180,E1 -5511.839,E2 -5511.839} C_VEL
LIN {X 0,Y 509.884,Z 261.786,A -85,B 0,C 180,E1 -5512.141,E2 -5512.141} C_VEL
LIN {X 0,Y 509.787,Z 261.797,A -85,B 0,C 180,E1 -5515.302,E2 -5515.302} C_VEL
LIN {X 0,Y 509.816,Z 261.792,A -85,B 0,C 180,E1 -5518.081,E2 -5518.081} C_VEL
LIN {X 0,Y 509.821,Z 261.792,A -85,B 0,C 180,E1 -5521.273,E2 -5521.273} C_VEL
LIN {X 0,Y 509.774,Z 261.795,A -85,B 0,C 180,E1 -5524.187,E2 -5524.187} C_VEL
LIN {X 0,Y 509.771,Z 261.797,A -85,B 0,C 180,E1 -5527.346,E2 -5527.346} C_VEL
LIN {X 0,Y 509.798,Z 261.791,A -85,B 0,C 180,E1 -5530.387,E2 -5530.387} C_VEL
LIN {X 0,Y 509.804,Z 261.791,A -85,B 0,C 180,E1 -5533.575,E2 -5533.575} C_VEL
LIN {X 0,Y 509.806,Z 261.79,A -85,B 0,C 180,E1 -5536.424,E2 -5536.424} C_VEL
LIN {X 0,Y 509.827,Z 261.786,A -85,B 0,C 180,E1 -5539.614,E2 -5539.614} C_VEL
LIN {X 0,Y 509.818,Z 261.79,A -85,B 0,C 180,E1 -5542.657,E2 -5542.657} C_VEL
LIN {X 0,Y 509.853,Z 261.784,A -85,B 0,C 180,E1 -5545.799,E2 -5545.799} C_VEL
LIN {X 0,Y 509.859,Z 261.788,A -85,B 0,C 180,E1 -5548.719,E2 -5548.719} C_VEL
LIN {X 0,Y 509.863,Z 261.791,A -85,B 0,C 180,E1 -5551.152,E2 -5551.152} C_VEL
LIN {X 0,Y 509.879,Z 261.784,A -85,B 0,C 180,E1 -5553.825,E2 -5553.825} C_VEL
LIN {X 0,Y 509.834,Z 261.789,A -85,B 0,C 180,E1 -5556.434,E2 -5556.434} C_VEL
LIN {X 0,Y 509.93,Z 261.776,A -85,B 0,C 180,E1 -5559.842,E2 -5559.842} C_VEL
LIN {X 0,Y 510.002,Z 261.774,A -85,B 0,C 180,E1 -5563.176,E2 -5563.176} C_VEL
LIN {X 0,Y 509.912,Z 261.899,A -85,B 0,C 180,E1 -5564.562,E2 -5564.562} C_VEL
LIN {X 0,Y 509.538,Z 277.778,A -85,B 0,C 180,E1 -5566.842,E2 -5566.842} C_VEL
LIN {X 0,Y 509.597,Z 283.991,A -85,B 0,C 180,E1 -5567.794,E2 -5567.794} C_VEL
LIN {X 0,Y 511.045,Z 295.495,A -85,B 0,C 180,E1 -5568.016,E2 -5568.016} C_VEL
LIN {X 0,Y 510.676,Z 362.104,A -85,B 0,C 180,E1 -5569.039,E2 -5569.039} C_VEL
LIN {X 0,Y 510.548,Z 372.495,A -85,B 0,C 180,E1 -5569.312,E2 -5569.312} C_VEL
LIN {X 0,Y 510.361,Z 384.198,A -85,B 0,C 180,E1 -5569.784,E2 -5569.784} C_VEL
LIN {X 0,Y 510.211,Z 393.1,A -85,B 0,C 180,E1 -5570.282,E2 -5570.282} C_VEL
LIN {X 0,Y 510.087,Z 401.56,A -85,B 0,C 180,E1 -5570.88,E2 -5570.88} C_VEL
LIN {X 0,Y 509.912,Z 409.54,A -85,B 0,C 180,E1 -5571.576,E2 -5571.576} C_VEL
LIN {X 0,Y 509.729,Z 416.12,A -85,B 0,C 180,E1 -5572.271,E2 -5572.271} C_VEL
LIN {X 0,Y 509.571,Z 422.237,A -85,B 0,C 180,E1 -5573.048,E2 -5573.048} C_VEL
LIN {X 0,Y 509.585,Z 427.532,A -85,B 0,C 180,E1 -5573.861,E2 -5573.861} C_VEL
LIN {X 0,Y 509.386,Z 430.88,A -85,B 0,C 180,E1 -5574.454,E2 -5574.454} C_VEL
LIN {X 0,Y 509.304,Z 434.64,A -85,B 0,C 180,E1 -5575.247,E2 -5575.247} C_VEL
LIN {X 0,Y 509.316,Z 438.892,A -85,B 0,C 180,E1 -5576.436,E2 -5576.436} C_VEL
LIN {X 0,Y 509.2,Z 441.865,A -85,B 0,C 180,E1 -5577.623,E2 -5577.623} C_VEL
LIN {X 0,Y 509.114,Z 443.177,A -85,B 0,C 180,E1 -5578.414,E2 -5578.414} C_VEL
LIN {X 0,Y 509.078,Z 444.003,A -85,B 0,C 180,E1 -5579.205,E2 -5579.205} C_VEL
LIN {X 0,Y 509.074,Z 444.306,A -85,B 0,C 180,E1 -5579.996,E2 -5579.996} C_VEL
LIN {X 0,Y 509.079,Z 444.024,A -85,B 0,C 180,E1 -5580.787,E2 -5580.787} C_VEL
LIN {X 0,Y 509.113,Z 443.263,A -85,B 0,C 180,E1 -5581.578,E2 -5581.578} C_VEL
LIN {X 0,Y 509.2,Z 442.02,A -85,B 0,C 180,E1 -5582.369,E2 -5582.369} C_VEL
LIN {X 0,Y 509.301,Z 439.11,A -85,B 0,C 180,E1 -5583.556,E2 -5583.556} C_VEL
LIN {X 0,Y 509.332,Z 436.46,A -85,B 0,C 180,E1 -5584.348,E2 -5584.348} C_VEL
LIN {X 0,Y 509.38,Z 431.263,A -85,B 0,C 180,E1 -5585.538,E2 -5585.538} C_VEL
LIN {X 0,Y 509.612,Z 425.559,A -85,B 0,C 180,E1 -5586.545,E2 -5586.545} C_VEL
LIN {X 0,Y 509.675,Z 418.583,A -85,B 0,C 180,E1 -5587.523,E2 -5587.523} C_VEL
LIN {X 0,Y 509.859,Z 410.47,A -85,B 0,C 180,E1 -5588.417,E2 -5588.417} C_VEL
LIN {X 0,Y 510.065,Z 402.722,A -85,B 0,C 180,E1 -5589.113,E2 -5589.113} C_VEL
LIN {X 0,Y 510.206,Z 394.568,A -85,B 0,C 180,E1 -5589.71,E2 -5589.71} C_VEL
LIN {X 0,Y 510.379,Z 386.088,A -85,B 0,C 180,E1 -5590.207,E2 -5590.207} C_VEL
LIN {X 0,Y 510.565,Z 376.188,A -85,B 0,C 180,E1 -5590.655,E2 -5590.655} C_VEL
LIN {X 0,Y 510.689,Z 363.924,A -85,B 0,C 180,E1 -5591.028,E2 -5591.028} C_VEL
LIN {X 0,Y 510.87,Z 342.385,A -85,B 0,C 180,E1 -5591.374,E2 -5591.374} C_VEL
LIN {X 0,Y 510.93,Z 293.802,A -85,B 0,C 180,E1 -5592.108,E2 -5592.108} C_VEL
LIN {X 0,Y 509.679,Z 285.8,A -85,B 0,C 180,E1 -5592.268,E2 -5592.268} C_VEL
LIN {X 0,Y 509.856,Z 271.878,A -85,B 0,C 180,E1 -5595.546,E2 -5595.546} C_VEL
LIN {X 0,Y 509.976,Z 262.14,A -85,B 0,C 180,E1 -5597.889,E2 -5597.889} C_VEL
LIN {X 0,Y 509.916,Z 261.781,A -85,B 0,C 180,E1 -5598.008,E2 -5598.008} C_VEL
LIN {X 0,Y 509.831,Z 261.793,A -85,B 0,C 180,E1 -5600.997,E2 -5600.997} C_VEL
LIN {X 0,Y 509.802,Z 261.794,A -85,B 0,C 180,E1 -5603.559,E2 -5603.559} C_VEL
LIN {X 0,Y 509.799,Z 261.791,A -85,B 0,C 180,E1 -5606.351,E2 -5606.351} C_VEL
LIN {X 0,Y 509.816,Z 261.793,A -85,B 0,C 180,E1 -5608.842,E2 -5608.842} C_VEL
LIN {X 0,Y 509.79,Z 261.798,A -85,B 0,C 180,E1 -5611.586,E2 -5611.586} C_VEL
LIN {X 0,Y 509.821,Z 261.788,A -85,B 0,C 180,E1 -5614.409,E2 -5614.409} C_VEL
LIN {X 0,Y 509.779,Z 261.796,A -85,B 0,C 180,E1 -5617.604,E2 -5617.604} C_VEL
LIN {X 0,Y 509.803,Z 261.791,A -85,B 0,C 180,E1 -5620.378,E2 -5620.378} C_VEL
LIN {X 0,Y 509.795,Z 261.793,A -85,B 0,C 180,E1 -5621.037,E2 -5621.037} C_VEL
LIN {X 0,Y 509.136,Z 261.88,A -85,B 0,C 180,E1 -5621.697,E2 -5621.697} C_VEL
LIN {X 0,Y 506.265,Z 262.238,A -85,B 0,C 180,E1 -5622.767,E2 -5622.767} C_VEL
LIN {X 0,Y 503.843,Z 262.538,A -85,B 0,C 180,E1 -5623.63,E2 -5623.63} C_VEL
LIN {X 0,Y 502.823,Z 262.662,A -85,B 0,C 180,E1 -5624.297,E2 -5624.297} C_VEL
LIN {X 0,Y 502.751,Z 262.669,A -85,B 0,C 180,E1 -5624.522,E2 -5624.522} C_VEL
LIN {X 0,Y 502.759,Z 262.673,A -85,B 0,C 180,E1 -5627.856,E2 -5627.856} C_VEL
LIN {X 0,Y 502.761,Z 262.668,A -85,B 0,C 180,E1 -5631.019,E2 -5631.019} C_VEL
LIN {X 0,Y 502.74,Z 262.676,A -85,B 0,C 180,E1 -5634.163,E2 -5634.163} C_VEL
LIN {X 0,Y 502.788,Z 262.665,A -85,B 0,C 180,E1 -5636.989,E2 -5636.989} C_VEL
LIN {X 0,Y 502.769,Z 262.672,A -85,B 0,C 180,E1 -5640.06,E2 -5640.06} C_VEL
LIN {X 0,Y 502.785,Z 262.669,A -85,B 0,C 180,E1 -5642.529,E2 -5642.529} C_VEL
LIN {X 0,Y 502.779,Z 262.666,A -85,B 0,C 180,E1 -5645.294,E2 -5645.294} C_VEL
LIN {X 0,Y 502.727,Z 262.675,A -85,B 0,C 180,E1 -5647.823,E2 -5647.823} C_VEL
LIN {X 0,Y 502.771,Z 262.672,A -85,B 0,C 180,E1 -5650.397,E2 -5650.397} C_VEL
LIN {X 0,Y 502.778,Z 262.668,A -85,B 0,C 180,E1 -5652.929,E2 -5652.929} C_VEL
LIN {X 0,Y 502.788,Z 262.665,A -85,B 0,C 180,E1 -5655.426,E2 -5655.426} C_VEL
LIN {X 0,Y 502.84,Z 262.663,A -85,B 0,C 180,E1 -5658.715,E2 -5658.715} C_VEL
LIN {X 0,Y 502.843,Z 262.659,A -85,B 0,C 180,E1 -5661.964,E2 -5661.964} C_VEL
LIN {X 0,Y 502.903,Z 262.654,A -85,B 0,C 180,E1 -5664.385,E2 -5664.385} C_VEL
LIN {X 0,Y 502.967,Z 262.643,A -85,B 0,C 180,E1 -5667.596,E2 -5667.596} C_VEL
LIN {X 0,Y 502.961,Z 262.643,A -85,B 0,C 180,E1 -5669.999,E2 -5669.999} C_VEL
LIN {X 0,Y 502.966,Z 262.644,A -85,B 0,C 180,E1 -5672.401,E2 -5672.401} C_VEL
LIN {X 0,Y 502.9,Z 262.652,A -85,B 0,C 180,E1 -5675.612,E2 -5675.612} C_VEL
LIN {X 0,Y 502.844,Z 262.658,A -85,B 0,C 180,E1 -5678.033,E2 -5678.033} C_VEL
LIN {X 0,Y 502.84,Z 262.663,A -85,B 0,C 180,E1 -5681.282,E2 -5681.282} C_VEL
LIN {X 0,Y 502.783,Z 262.666,A -85,B 0,C 180,E1 -5684.571,E2 -5684.571} C_VEL
LIN {X 0,Y 502.799,Z 262.665,A -85,B 0,C 180,E1 -5687.908,E2 -5687.908} C_VEL
LIN {X 0,Y 502.767,Z 262.667,A -85,B 0,C 180,E1 -5690.537,E2 -5690.537} C_VEL
LIN {X 0,Y 502.741,Z 262.673,A -85,B 0,C 180,E1 -5693.041,E2 -5693.041} C_VEL
LIN {X 0,Y 502.787,Z 262.67,A -85,B 0,C 180,E1 -5695.677,E2 -5695.677} C_VEL
LIN {X 0,Y 502.783,Z 262.666,A -85,B 0,C 180,E1 -5698.374,E2 -5698.374} C_VEL
LIN {X 0,Y 502.739,Z 262.676,A -85,B 0,C 180,E1 -5701.502,E2 -5701.502} C_VEL
LIN {X 0,Y 502.75,Z 262.671,A -85,B 0,C 180,E1 -5704.447,E2 -5704.447} C_VEL
LIN {X 0,Y 502.726,Z 262.673,A -85,B 0,C 180,E1 -5707.181,E2 -5707.181} C_VEL
LIN {X 0,Y 502.79,Z 262.669,A -85,B 0,C 180,E1 -5710.013,E2 -5710.013} C_VEL
LIN {X 0,Y 502.775,Z 262.671,A -85,B 0,C 180,E1 -5712.205,E2 -5712.205} C_VEL
LIN {X 0,Y 502.75,Z 262.671,A -85,B 0,C 180,E1 -5715.471,E2 -5715.471} C_VEL
LIN {X 0,Y 502.781,Z 262.67,A -85,B 0,C 180,E1 -5717.868,E2 -5717.868} C_VEL
LIN {X 0,Y 502.763,Z 262.668,A -85,B 0,C 180,E1 -5721.028,E2 -5721.028} C_VEL
LIN {X 0,Y 502.742,Z 262.676,A -85,B 0,C 180,E1 -5724.171,E2 -5724.171} C_VEL
LIN {X 0,Y 502.791,Z 262.666,A -85,B 0,C 180,E1 -5726.997,E2 -5726.997} C_VEL
LIN {X 0,Y 502.775,Z 262.669,A -85,B 0,C 180,E1 -5730.069,E2 -5730.069} C_VEL
LIN {X 0,Y 502.788,Z 262.67,A -85,B 0,C 180,E1 -5732.537,E2 -5732.537} C_VEL
LIN {X 0,Y 502.742,Z 262.671,A -85,B 0,C 180,E1 -5735.315,E2 -5735.315} C_VEL
LIN {X 0,Y 502.745,Z 262.67,A -85,B 0,C 180,E1 -5737.831,E2 -5737.831} C_VEL
LIN {X 0,Y 502.787,Z 262.668,A -85,B 0,C 180,E1 -5740.404,E2 -5740.404} C_VEL
LIN {X 0,Y 502.784,Z 262.67,A -85,B 0,C 180,E1 -5742.935,E2 -5742.935} C_VEL
LIN {X 0,Y 502.812,Z 262.664,A -85,B 0,C 180,E1 -5745.433,E2 -5745.433} C_VEL
LIN {X 0,Y 502.849,Z 262.662,A -85,B 0,C 180,E1 -5748.721,E2 -5748.721} C_VEL
LIN {X 0,Y 502.855,Z 262.656,A -85,B 0,C 180,E1 -5751.97,E2 -5751.97} C_VEL
LIN {X 0,Y 502.9,Z 262.651,A -85,B 0,C 180,E1 -5754.39,E2 -5754.39} C_VEL
LIN {X 0,Y 502.993,Z 262.643,A -85,B 0,C 180,E1 -5757.602,E2 -5757.602} C_VEL
LIN {X 0,Y 502.983,Z 262.641,A -85,B 0,C 180,E1 -5760.004,E2 -5760.004} C_VEL
LIN {X 0,Y 502.996,Z 262.639,A -85,B 0,C 180,E1 -5762.406,E2 -5762.406} C_VEL
LIN {X 0,Y 502.899,Z 262.656,A -85,B 0,C 180,E1 -5765.618,E2 -5765.618} C_VEL
LIN {X 0,Y 502.847,Z 262.658,A -85,B 0,C 180,E1 -5768.847,E2 -5768.847} C_VEL
LIN {X 0,Y 502.832,Z 262.662,A -85,B 0,C 180,E1 -5772.105,E2 -5772.105} C_VEL
LIN {X 0,Y 502.835,Z 262.663,A -85,B 0,C 180,E1 -5775.403,E2 -5775.403} C_VEL
LIN {X 0,Y 502.8,Z 262.663,A -85,B 0,C 180,E1 -5778.756,E2 -5778.756} C_VEL
LIN {X 0,Y 502.77,Z 262.669,A -85,B 0,C 180,E1 -5781.315,E2 -5781.315} C_VEL
LIN {X 0,Y 502.759,Z 262.674,A -85,B 0,C 180,E1 -5783.918,E2 -5783.918} C_VEL
LIN {X 0,Y 502.777,Z 262.668,A -85,B 0,C 180,E1 -5786.574,E2 -5786.574} C_VEL
LIN {X 0,Y 502.806,Z 262.663,A -85,B 0,C 180,E1 -5789.292,E2 -5789.292} C_VEL
LIN {X 0,Y 502.777,Z 262.672,A -85,B 0,C 180,E1 -5792.088,E2 -5792.088} C_VEL
LIN {X 0,Y 502.782,Z 262.666,A -85,B 0,C 180,E1 -5794.97,E2 -5794.97} C_VEL
LIN {X 0,Y 502.758,Z 262.673,A -85,B 0,C 180,E1 -5798.484,E2 -5798.484} C_VEL
LIN {X 0,Y 502.76,Z 262.669,A -85,B 0,C 180,E1 -5801.074,E2 -5801.074} C_VEL
LIN {X 0,Y 502.776,Z 262.672,A -85,B 0,C 180,E1 -5804.343,E2 -5804.343} C_VEL
LIN {X 0,Y 502.737,Z 262.676,A -85,B 0,C 180,E1 -5806.768,E2 -5806.768} C_VEL
LIN {X 0,Y 502.769,Z 262.668,A -85,B 0,C 180,E1 -5809.985,E2 -5809.985} C_VEL
LIN {X 0,Y 502.749,Z 262.674,A -85,B 0,C 180,E1 -5813.053,E2 -5813.053} C_VEL
LIN {X 0,Y 502.784,Z 262.665,A -85,B 0,C 180,E1 -5816.007,E2 -5816.007} C_VEL
LIN {X 0,Y 502.784,Z 262.671,A -85,B 0,C 180,E1 -5818.858,E2 -5818.858} C_VEL
LIN {X 0,Y 502.77,Z 262.667,A -85,B 0,C 180,E1 -5821.723,E2 -5821.723} C_VEL
LIN {X 0,Y 502.769,Z 262.668,A -85,B 0,C 180,E1 -5824.322,E2 -5824.322} C_VEL
LIN {X 0,Y 502.802,Z 262.737,A -85,B 0,C 180,E1 -5826.553,E2 -5826.553} C_VEL
LIN {X 0,Y 503.904,Z 269.331,A -85,B 0,C 180,E1 -5827.88,E2 -5827.88} C_VEL
LIN {X 0,Y 503.648,Z 282.753,A -85,B 0,C 180,E1 -5830.435,E2 -5830.435} C_VEL
LIN {X 0,Y 503.139,Z 299.542,A -85,B 0,C 180,E1 -5833.571,E2 -5833.571} C_VEL
LIN {X 0,Y 502.786,Z 316.304,A -85,B 0,C 180,E1 -5836.667,E2 -5836.667} C_VEL
LIN {X 0,Y 502.693,Z 321.267,A -85,B 0,C 180,E1 -5837.578,E2 -5837.578} C_VEL
LIN {X 0,Y 504.074,Z 333.287,A -85,B 0,C 180,E1 -5837.817,E2 -5837.817} C_VEL
LIN {X 0,Y 503.7,Z 399.456,A -85,B 0,C 180,E1 -5838.839,E2 -5838.839} C_VEL
LIN {X 0,Y 503.473,Z 410.412,A -85,B 0,C 180,E1 -5839.139,E2 -5839.139} C_VEL
LIN {X 0,Y 503.251,Z 422.091,A -85,B 0,C 180,E1 -5839.643,E2 -5839.643} C_VEL
LIN {X 0,Y 503.08,Z 430.793,A -85,B 0,C 180,E1 -5840.148,E2 -5840.148} C_VEL
LIN {X 0,Y 502.913,Z 439.126,A -85,B 0,C 180,E1 -5840.754,E2 -5840.754} C_VEL
LIN {X 0,Y 502.712,Z 447.023,A -85,B 0,C 180,E1 -5841.459,E2 -5841.459} C_VEL
LIN {X 0,Y 502.523,Z 453.55,A -85,B 0,C 180,E1 -5842.164,E2 -5842.164} C_VEL
LIN {X 0,Y 502.431,Z 459.913,A -85,B 0,C 180,E1 -5842.991,E2 -5842.991} C_VEL
LIN {X 0,Y 502.305,Z 466.114,A -85,B 0,C 180,E1 -5843.978,E2 -5843.978} C_VEL
LIN {X 0,Y 502.145,Z 471.987,A -85,B 0,C 180,E1 -5845.184,E2 -5845.184} C_VEL
LIN {X 0,Y 502.154,Z 475.044,A -85,B 0,C 180,E1 -5845.989,E2 -5845.989} C_VEL
LIN {X 0,Y 502.135,Z 477.414,A -85,B 0,C 180,E1 -5846.792,E2 -5846.792} C_VEL
LIN {X 0,Y 502.095,Z 479.208,A -85,B 0,C 180,E1 -5847.595,E2 -5847.595} C_VEL
LIN {X 0,Y 502.037,Z 480.49,A -85,B 0,C 180,E1 -5848.397,E2 -5848.397} C_VEL
LIN {X 0,Y 501.991,Z 481.285,A -85,B 0,C 180,E1 -5849.199,E2 -5849.199} C_VEL
LIN {X 0,Y 501.984,Z 481.574,A -85,B 0,C 180,E1 -5850.001,E2 -5850.001} C_VEL
LIN {X 0,Y 501.991,Z 481.262,A -85,B 0,C 180,E1 -5850.804,E2 -5850.804} C_VEL
LIN {X 0,Y 502.037,Z 480.451,A -85,B 0,C 180,E1 -5851.606,E2 -5851.606} C_VEL
LIN {X 0,Y 502.096,Z 479.151,A -85,B 0,C 180,E1 -5852.408,E2 -5852.408} C_VEL
LIN {X 0,Y 502.166,Z 476.148,A -85,B 0,C 180,E1 -5853.612,E2 -5853.612} C_VEL
LIN {X 0,Y 502.133,Z 473.404,A -85,B 0,C 180,E1 -5854.416,E2 -5854.416} C_VEL
LIN {X 0,Y 502.262,Z 468.06,A -85,B 0,C 180,E1 -5855.622,E2 -5855.622} C_VEL
LIN {X 0,Y 502.378,Z 461.241,A -85,B 0,C 180,E1 -5856.79,E2 -5856.79} C_VEL
LIN {X 0,Y 502.477,Z 454.973,A -85,B 0,C 180,E1 -5857.637,E2 -5857.637} C_VEL
LIN {X 0,Y 502.661,Z 447.683,A -85,B 0,C 180,E1 -5858.443,E2 -5858.443} C_VEL
LIN {X 0,Y 502.849,Z 439.903,A -85,B 0,C 180,E1 -5859.149,E2 -5859.149} C_VEL
LIN {X 0,Y 503.012,Z 431.732,A -85,B 0,C 180,E1 -5859.755,E2 -5859.755} C_VEL
LIN {X 0,Y 503.166,Z 423.268,A -85,B 0,C 180,E1 -5860.26,E2 -5860.26} C_VEL
LIN {X 0,Y 503.411,Z 413.442,A -85,B 0,C 180,E1 -5860.712,E2 -5860.712} C_VEL
LIN {X 0,Y 503.651,Z 401.735,A -85,B 0,C 180,E1 -5861.089,E2 -5861.089} C_VEL
LIN {X 0,Y 503.787,Z 382.591,A -85,B 0,C 180,E1 -5861.415,E2 -5861.415} C_VEL
LIN {X 0,Y 503.96,Z 331.85,A -85,B 0,C 180,E1 -5862.199,E2 -5862.199} C_VEL
LIN {X 0,Y 502.603,Z 320.382,A -85,B 0,C 180,E1 -5862.419,E2 -5862.419} C_VEL
LIN {X 0,Y 502.824,Z 302.925,A -85,B 0,C 180,E1 -5865.402,E2 -5865.402} C_VEL
LIN {X 0,Y 503.008,Z 286.525,A -85,B 0,C 180,E1 -5868.175,E2 -5868.175} C_VEL
LIN {X 0,Y 503.179,Z 270.257,A -85,B 0,C 180,E1 -5870.909,E2 -5870.909} C_VEL
LIN {X 0,Y 503.027,Z 264.057,A -85,B 0,C 180,E1 -5871.947,E2 -5871.947} C_VEL
LIN {X 0,Y 502.849,Z 262.663,A -85,B 0,C 180,E1 -5872.21,E2 -5872.21} C_VEL
LIN {X 0,Y 502.764,Z 262.67,A -85,B 0,C 180,E1 -5875.681,E2 -5875.681} C_VEL
LIN {X 0,Y 502.769,Z 262.672,A -85,B 0,C 180,E1 -5878.378,E2 -5878.378} C_VEL
LIN {X 0,Y 502.77,Z 262.668,A -85,B 0,C 180,E1 -5881.492,E2 -5881.492} C_VEL
LIN {X 0,Y 502.727,Z 262.675,A -85,B 0,C 180,E1 -5884.429,E2 -5884.429} C_VEL
LIN {X 0,Y 502.726,Z 262.677,A -85,B 0,C 180,E1 -5887.168,E2 -5887.168} C_VEL
LIN {X 0,Y 502.743,Z 262.668,A -85,B 0,C 180,E1 -5890.021,E2 -5890.021} C_VEL
LIN {X 0,Y 502.75,Z 262.673,A -85,B 0,C 180,E1 -5893.235,E2 -5893.235} C_VEL
LIN {X 0,Y 502.781,Z 262.665,A -85,B 0,C 180,E1 -5895.658,E2 -5895.658} C_VEL
LIN {X 0,Y 502.777,Z 262.672,A -85,B 0,C 180,E1 -5899.012,E2 -5899.012} C_VEL
LIN {X 0,Y 502.784,Z 262.662,A -85,B 0,C 180,E1 -5902.043,E2 -5902.043} C_VEL
LIN {X 0,Y 502.802,Z 262.669,A -85,B 0,C 180,E1 -5905.032,E2 -5905.032} C_VEL
LIN {X 0,Y 502.796,Z 262.664,A -85,B 0,C 180,E1 -5907.914,E2 -5907.914} C_VEL
LIN {X 0,Y 502.825,Z 262.664,A -85,B 0,C 180,E1 -5910.709,E2 -5910.709} C_VEL
LIN {X 0,Y 502.814,Z 262.667,A -85,B 0,C 180,E1 -5913.452,E2 -5913.452} C_VEL
LIN {X 0,Y 502.785,Z 262.667,A -85,B 0,C 180,E1 -5916.083,E2 -5916.083} C_VEL
LIN {X 0,Y 502.797,Z 262.668,A -85,B 0,C 180,E1 -5918.686,E2 -5918.686} C_VEL
LIN {X 0,Y 502.84,Z 262.666,A -85,B 0,C 180,E1 -5921.245,E2 -5921.245} C_VEL
LIN {X 0,Y 502.966,Z 262.65,A -85,B 0,C 180,E1 -5924.393,E2 -5924.393} C_VEL
LIN {X 0,Y 502.862,Z 262.91,A -85,B 0,C 180,E1 -5924.546,E2 -5924.546} C_VEL
LIN {X 0,Y 502.527,Z 279.127,A -85,B 0,C 180,E1 -5926.861,E2 -5926.861} C_VEL
LIN {X 0,Y 502.595,Z 284.232,A -85,B 0,C 180,E1 -5927.621,E2 -5927.621} C_VEL
LIN {X 0,Y 504.152,Z 296.954,A -85,B 0,C 180,E1 -5927.865,E2 -5927.865} C_VEL
LIN {X 0,Y 503.696,Z 363.032,A -85,B 0,C 180,E1 -5928.91,E2 -5928.91} C_VEL
LIN {X 0,Y 503.576,Z 374.729,A -85,B 0,C 180,E1 -5929.238,E2 -5929.238} C_VEL
LIN {X 0,Y 503.347,Z 386.078,A -85,B 0,C 180,E1 -5929.742,E2 -5929.742} C_VEL
LIN {X 0,Y 503.17,Z 394.656,A -85,B 0,C 180,E1 -5930.246,E2 -5930.246} C_VEL
LIN {X 0,Y 503.052,Z 402.881,A -85,B 0,C 180,E1 -5930.852,E2 -5930.852} C_VEL
LIN {X 0,Y 502.843,Z 410.684,A -85,B 0,C 180,E1 -5931.558,E2 -5931.558} C_VEL
LIN {X 0,Y 502.635,Z 419.652,A -85,B 0,C 180,E1 -5932.565,E2 -5932.565} C_VEL
LIN {X 0,Y 502.572,Z 426.549,A -85,B 0,C 180,E1 -5933.573,E2 -5933.573} C_VEL
LIN {X 0,Y 502.341,Z 431.094,A -85,B 0,C 180,E1 -5934.376,E2 -5934.376} C_VEL
LIN {X 0,Y 502.222,Z 434.869,A -85,B 0,C 180,E1 -5935.18,E2 -5935.18} C_VEL
LIN {X 0,Y 502.232,Z 439.137,A -85,B 0,C 180,E1 -5936.386,E2 -5936.386} C_VEL
LIN {X 0,Y 502.134,Z 442.12,A -85,B 0,C 180,E1 -5937.59,E2 -5937.59} C_VEL
LIN {X 0,Y 502.038,Z 443.437,A -85,B 0,C 180,E1 -5938.392,E2 -5938.392} C_VEL
LIN {X 0,Y 501.995,Z 444.266,A -85,B 0,C 180,E1 -5939.194,E2 -5939.194} C_VEL
LIN {X 0,Y 501.988,Z 444.568,A -85,B 0,C 180,E1 -5939.996,E2 -5939.996} C_VEL
LIN {X 0,Y 501.996,Z 444.283,A -85,B 0,C 180,E1 -5940.798,E2 -5940.798} C_VEL
LIN {X 0,Y 502.037,Z 443.517,A -85,B 0,C 180,E1 -5941.6,E2 -5941.6} C_VEL
LIN {X 0,Y 502.134,Z 442.265,A -85,B 0,C 180,E1 -5942.402,E2 -5942.402} C_VEL
LIN {X 0,Y 502.219,Z 439.341,A -85,B 0,C 180,E1 -5943.606,E2 -5943.606} C_VEL
LIN {X 0,Y 502.261,Z 436.676,A -85,B 0,C 180,E1 -5944.41,E2 -5944.41} C_VEL
LIN {X 0,Y 502.335,Z 431.452,A -85,B 0,C 180,E1 -5945.616,E2 -5945.616} C_VEL
LIN {X 0,Y 502.565,Z 426.198,A -85,B 0,C 180,E1 -5946.558,E2 -5946.558} C_VEL
LIN {X 0,Y 502.627,Z 418.704,A -85,B 0,C 180,E1 -5947.629,E2 -5947.629} C_VEL
LIN {X 0,Y 502.836,Z 410.556,A -85,B 0,C 180,E1 -5948.536,E2 -5948.536} C_VEL
LIN {X 0,Y 503.04,Z 402.767,A -85,B 0,C 180,E1 -5949.241,E2 -5949.241} C_VEL
LIN {X 0,Y 503.215,Z 394.565,A -85,B 0,C 180,E1 -5949.846,E2 -5949.846} C_VEL
LIN {X 0,Y 503.413,Z 384.154,A -85,B 0,C 180,E1 -5950.452,E2 -5950.452} C_VEL
LIN {X 0,Y 503.635,Z 372.467,A -85,B 0,C 180,E1 -5950.93,E2 -5950.93} C_VEL
LIN {X 0,Y 503.738,Z 362.123,A -85,B 0,C 180,E1 -5951.208,E2 -5951.208} C_VEL
LIN {X 0,Y 504.03,Z 294.741,A -85,B 0,C 180,E1 -5952.259,E2 -5952.259} C_VEL
LIN {X 0,Y 502.656,Z 286.033,A -85,B 0,C 180,E1 -5952.433,E2 -5952.433} C_VEL
LIN {X 0,Y 502.858,Z 271.818,A -85,B 0,C 180,E1 -5955.81,E2 -5955.81} C_VEL
LIN {X 0,Y 502.958,Z 263.23,A -85,B 0,C 180,E1 -5957.898,E2 -5957.898} C_VEL
LIN {X 0,Y 502.861,Z 262.66,A -85,B 0,C 180,E1 -5958.125,E2 -5958.125} C_VEL
LIN {X 0,Y 502.766,Z 262.673,A -85,B 0,C 180,E1 -5961.306,E2 -5961.306} C_VEL
LIN {X 0,Y 502.75,Z 262.67,A -85,B 0,C 180,E1 -5963.91,E2 -5963.91} C_VEL
LIN {X 0,Y 502.766,Z 262.669,A -85,B 0,C 180,E1 -5966.566,E2 -5966.566} C_VEL
LIN {X 0,Y 502.789,Z 262.666,A -85,B 0,C 180,E1 -5969.928,E2 -5969.928} C_VEL
LIN {X 0,Y 502.808,Z 262.667,A -85,B 0,C 180,E1 -5973.026,E2 -5973.026} C_VEL
LIN {X 0,Y 502.741,Z 262.673,A -85,B 0,C 180,E1 -5975.947,E2 -5975.947} C_VEL
LIN {X 0,Y 502.769,Z 262.669,A -85,B 0,C 180,E1 -5978.971,E2 -5978.971} C_VEL
LIN {X 0,Y 502.771,Z 262.668,A -85,B 0,C 180,E1 -5982.194,E2 -5982.194} C_VEL
LIN {X 0,Y 502.751,Z 262.669,A -85,B 0,C 180,E1 -5984.522,E2 -5984.522} C_VEL
LIN {X 0,Y 502.105,Z 262.754,A -85,B 0,C 180,E1 -5985.191,E2 -5985.191} C_VEL
LIN {X 0,Y 499.232,Z 263.109,A -85,B 0,C 180,E1 -5986.275,E2 -5986.275} C_VEL
LIN {X 0,Y 496.802,Z 263.413,A -85,B 0,C 180,E1 -5987.149,E2 -5987.149} C_VEL
LIN {X 0,Y 495.779,Z 263.542,A -85,B 0,C 180,E1 -5987.825,E2 -5987.825} C_VEL
LIN {X 0,Y 495.709,Z 263.549,A -85,B 0,C 180,E1 -5988.054,E2 -5988.054} C_VEL
LIN {X 0,Y 495.722,Z 263.546,A -85,B 0,C 180,E1 -5991.227,E2 -5991.227} C_VEL
LIN {X 0,Y 495.712,Z 263.548,A -85,B 0,C 180,E1 -5994.458,E2 -5994.458} C_VEL
LIN {X 0,Y 495.723,Z 263.546,A -85,B 0,C 180,E1 -5997.401,E2 -5997.401} C_VEL
LIN {X 0,Y 495.721,Z 263.55,A -85,B 0,C 180,E1 -6000.25,E2 -6000.25} C_VEL
LIN {X 0,Y 495.785,Z 263.537,A -85,B 0,C 180,E1 -6003.244,E2 -6003.244} C_VEL
LIN {X 0,Y 495.702,Z 263.55,A -85,B 0,C 180,E1 -6005.721,E2 -6005.721} C_VEL
LIN {X 0,Y 495.689,Z 263.554,A -85,B 0,C 180,E1 -6008.367,E2 -6008.367} C_VEL
LIN {X 0,Y 495.73,Z 263.546,A -85,B 0,C 180,E1 -6010.968,E2 -6010.968} C_VEL
LIN {X 0,Y 495.723,Z 263.545,A -85,B 0,C 180,E1 -6013.527,E2 -6013.527} C_VEL
LIN {X 0,Y 495.74,Z 263.546,A -85,B 0,C 180,E1 -6016.053,E2 -6016.053} C_VEL
LIN {X 0,Y 495.814,Z 263.538,A -85,B 0,C 180,E1 -6018.553,E2 -6018.553} C_VEL
LIN {X 0,Y 495.815,Z 263.534,A -85,B 0,C 180,E1 -6021.85,E2 -6021.85} C_VEL
LIN {X 0,Y 495.857,Z 263.531,A -85,B 0,C 180,E1 -6024.305,E2 -6024.305} C_VEL
LIN {X 0,Y 495.937,Z 263.519,A -85,B 0,C 180,E1 -6027.562,E2 -6027.562} C_VEL
LIN {X 0,Y 495.933,Z 263.519,A -85,B 0,C 180,E1 -6029.999,E2 -6029.999} C_VEL
LIN {X 0,Y 495.936,Z 263.521,A -85,B 0,C 180,E1 -6032.435,E2 -6032.435} C_VEL
LIN {X 0,Y 495.854,Z 263.53,A -85,B 0,C 180,E1 -6035.692,E2 -6035.692} C_VEL
LIN {X 0,Y 495.817,Z 263.533,A -85,B 0,C 180,E1 -6038.147,E2 -6038.147} C_VEL
LIN {X 0,Y 495.813,Z 263.538,A -85,B 0,C 180,E1 -6041.445,E2 -6041.445} C_VEL
LIN {X 0,Y 495.728,Z 263.547,A -85,B 0,C 180,E1 -6044.783,E2 -6044.783} C_VEL
LIN {X 0,Y 495.726,Z 263.549,A -85,B 0,C 180,E1 -6047.319,E2 -6047.319} C_VEL
LIN {X 0,Y 495.717,Z 263.548,A -85,B 0,C 180,E1 -6049.891,E2 -6049.891} C_VEL
LIN {X 0,Y 495.702,Z 263.549,A -85,B 0,C 180,E1 -6052.863,E2 -6052.863} C_VEL
LIN {X 0,Y 495.743,Z 263.545,A -85,B 0,C 180,E1 -6056.069,E2 -6056.069} C_VEL
LIN {X 0,Y 495.721,Z 263.545,A -85,B 0,C 180,E1 -6058.816,E2 -6058.816} C_VEL
LIN {X 0,Y 495.701,Z 263.552,A -85,B 0,C 180,E1 -6061.728,E2 -6061.728} C_VEL
LIN {X 0,Y 495.72,Z 263.545,A -85,B 0,C 180,E1 -6064.698,E2 -6064.698} C_VEL
LIN {X 0,Y 495.679,Z 263.555,A -85,B 0,C 180,E1 -6067.564,E2 -6067.564} C_VEL
LIN {X 0,Y 495.755,Z 263.545,A -85,B 0,C 180,E1 -6070.057,E2 -6070.057} C_VEL
LIN {X 0,Y 495.712,Z 263.546,A -85,B 0,C 180,E1 -6072.882,E2 -6072.882} C_VEL
LIN {X 0,Y 495.686,Z 263.555,A -85,B 0,C 180,E1 -6076.003,E2 -6076.003} C_VEL
LIN {X 0,Y 495.72,Z 263.548,A -85,B 0,C 180,E1 -6078.709,E2 -6078.709} C_VEL
LIN {X 0,Y 495.709,Z 263.547,A -85,B 0,C 180,E1 -6081.412,E2 -6081.412} C_VEL
LIN {X 0,Y 495.714,Z 263.55,A -85,B 0,C 180,E1 -6084.467,E2 -6084.467} C_VEL
LIN {X 0,Y 495.727,Z 263.544,A -85,B 0,C 180,E1 -6087.41,E2 -6087.41} C_VEL
LIN {X 0,Y 495.726,Z 263.55,A -85,B 0,C 180,E1 -6090.258,E2 -6090.258} C_VEL
LIN {X 0,Y 495.768,Z 263.54,A -85,B 0,C 180,E1 -6093.259,E2 -6093.259} C_VEL
LIN {X 0,Y 495.705,Z 263.552,A -85,B 0,C 180,E1 -6096.616,E2 -6096.616} C_VEL
LIN {X 0,Y 495.746,Z 263.544,A -85,B 0,C 180,E1 -6099.328,E2 -6099.328} C_VEL
LIN {X 0,Y 495.748,Z 263.542,A -85,B 0,C 180,E1 -6101.833,E2 -6101.833} C_VEL
LIN {X 0,Y 495.795,Z 263.54,A -85,B 0,C 180,E1 -6104.553,E2 -6104.553} C_VEL
LIN {X 0,Y 495.802,Z 263.535,A -85,B 0,C 180,E1 -6107.97,E2 -6107.97} C_VEL
LIN {X 0,Y 495.807,Z 263.539,A -85,B 0,C 180,E1 -6111.034,E2 -6111.034} C_VEL
LIN {X 0,Y 495.826,Z 263.536,A -85,B 0,C 180,E1 -6113.493,E2 -6113.493} C_VEL
LIN {X 0,Y 495.689,Z 263.55,A -85,B 0,C 180,E1 -6115.939,E2 -6115.939} C_VEL
LIN {X 0,Y 495.961,Z 263.52,A -85,B 0,C 180,E1 -6117.568,E2 -6117.568} C_VEL
LIN {X 0,Y 495.953,Z 263.517,A -85,B 0,C 180,E1 -6120.004,E2 -6120.004} C_VEL
LIN {X 0,Y 495.965,Z 263.515,A -85,B 0,C 180,E1 -6122.44,E2 -6122.44} C_VEL
LIN {X 0,Y 495.855,Z 263.533,A -85,B 0,C 180,E1 -6125.698,E2 -6125.698} C_VEL
LIN {X 0,Y 495.817,Z 263.535,A -85,B 0,C 180,E1 -6128.974,E2 -6128.974} C_VEL
LIN {X 0,Y 495.817,Z 263.537,A -85,B 0,C 180,E1 -6132.038,E2 -6132.038} C_VEL
LIN {X 0,Y 495.792,Z 263.541,A -85,B 0,C 180,E1 -6135.446,E2 -6135.446} C_VEL
LIN {X 0,Y 495.759,Z 263.541,A -85,B 0,C 180,E1 -6139.033,E2 -6139.033} C_VEL
LIN {X 0,Y 495.731,Z 263.549,A -85,B 0,C 180,E1 -6141.633,E2 -6141.633} C_VEL
LIN {X 0,Y 495.705,Z 263.552,A -85,B 0,C 180,E1 -6144.28,E2 -6144.28} C_VEL
LIN {X 0,Y 495.727,Z 263.544,A -85,B 0,C 180,E1 -6146.982,E2 -6146.982} C_VEL
LIN {X 0,Y 495.758,Z 263.545,A -85,B 0,C 180,E1 -6150.15,E2 -6150.15} C_VEL
LIN {X 0,Y 495.746,Z 263.542,A -85,B 0,C 180,E1 -6153.24,E2 -6153.24} C_VEL
LIN {X 0,Y 495.699,Z 263.554,A -85,B 0,C 180,E1 -6156.089,E2 -6156.089} C_VEL
LIN {X 0,Y 495.735,Z 263.547,A -85,B 0,C 180,E1 -6158.767,E2 -6158.767} C_VEL
LIN {X 0,Y 495.72,Z 263.546,A -85,B 0,C 180,E1 -6161.787,E2 -6161.787} C_VEL
LIN {X 0,Y 495.73,Z 263.545,A -85,B 0,C 180,E1 -6165.144,E2 -6165.144} C_VEL
LIN {X 0,Y 495.722,Z 263.548,A -85,B 0,C 180,E1 -6168.218,E2 -6168.218} C_VEL
LIN {X 0,Y 495.741,Z 263.545,A -85,B 0,C 180,E1 -6171.238,E2 -6171.238} C_VEL
LIN {X 0,Y 495.738,Z 263.547,A -85,B 0,C 180,E1 -6174.464,E2 -6174.464} C_VEL
LIN {X 0,Y 495.75,Z 263.544,A -85,B 0,C 180,E1 -6177.406,E2 -6177.406} C_VEL
LIN {X 0,Y 495.741,Z 263.543,A -85,B 0,C 180,E1 -6180.254,E2 -6180.254} C_VEL
LIN {X 0,Y 495.738,Z 263.547,A -85,B 0,C 180,E1 -6183.273,E2 -6183.273} C_VEL
LIN {X 0,Y 495.788,Z 263.649,A -85,B 0,C 180,E1 -6186.423,E2 -6186.423} C_VEL
LIN {X 0,Y 496.976,Z 271.386,A -85,B 0,C 180,E1 -6187.993,E2 -6187.993} C_VEL
LIN {X 0,Y 496.503,Z 287.023,A -85,B 0,C 180,E1 -6191.002,E2 -6191.002} C_VEL
LIN {X 0,Y 496.048,Z 302.666,A -85,B 0,C 180,E1 -6193.964,E2 -6193.964} C_VEL
LIN {X 0,Y 495.662,Z 319.31,A -85,B 0,C 180,E1 -6197.077,E2 -6197.077} C_VEL
LIN {X 0,Y 495.642,Z 321.081,A -85,B 0,C 180,E1 -6197.407,E2 -6197.407} C_VEL
LIN {X 0,Y 497.115,Z 334.856,A -85,B 0,C 180,E1 -6197.673,E2 -6197.673} C_VEL
LIN {X 0,Y 496.716,Z 398.521,A -85,B 0,C 180,E1 -6198.68,E2 -6198.68} C_VEL
LIN {X 0,Y 496.514,Z 408.886,A -85,B 0,C 180,E1 -6198.959,E2 -6198.959} C_VEL
LIN {X 0,Y 496.295,Z 419.641,A -85,B 0,C 180,E1 -6199.393,E2 -6199.393} C_VEL
LIN {X 0,Y 496.06,Z 430.327,A -85,B 0,C 180,E1 -6200.007,E2 -6200.007} C_VEL
LIN {X 0,Y 495.887,Z 438.702,A -85,B 0,C 180,E1 -6200.621,E2 -6200.621} C_VEL
LIN {X 0,Y 495.634,Z 446.629,A -85,B 0,C 180,E1 -6201.336,E2 -6201.336} C_VEL
LIN {X 0,Y 495.455,Z 453.186,A -85,B 0,C 180,E1 -6202.052,E2 -6202.052} C_VEL
LIN {X 0,Y 495.359,Z 459.573,A -85,B 0,C 180,E1 -6202.891,E2 -6202.891} C_VEL
LIN {X 0,Y 495.204,Z 466.945,A -85,B 0,C 180,E1 -6204.096,E2 -6204.096} C_VEL
LIN {X 0,Y 495.07,Z 471.696,A -85,B 0,C 180,E1 -6205.115,E2 -6205.115} C_VEL
LIN {X 0,Y 495.05,Z 474.76,A -85,B 0,C 180,E1 -6205.931,E2 -6205.931} C_VEL
LIN {X 0,Y 495.059,Z 477.139,A -85,B 0,C 180,E1 -6206.746,E2 -6206.746} C_VEL
LIN {X 0,Y 495.002,Z 478.941,A -85,B 0,C 180,E1 -6207.56,E2 -6207.56} C_VEL
LIN {X 0,Y 494.963,Z 480.229,A -85,B 0,C 180,E1 -6208.374,E2 -6208.374} C_VEL
LIN {X 0,Y 494.911,Z 481.026,A -85,B 0,C 180,E1 -6209.188,E2 -6209.188} C_VEL
LIN {X 0,Y 494.902,Z 481.314,A -85,B 0,C 180,E1 -6210.001,E2 -6210.001} C_VEL
LIN {X 0,Y 494.911,Z 480.999,A -85,B 0,C 180,E1 -6210.815,E2 -6210.815} C_VEL
LIN {X 0,Y 494.963,Z 480.18,A -85,B 0,C 180,E1 -6211.629,E2 -6211.629} C_VEL
LIN {X 0,Y 495.003,Z 478.868,A -85,B 0,C 180,E1 -6212.443,E2 -6212.443} C_VEL
LIN {X 0,Y 495.087,Z 475.85,A -85,B 0,C 180,E1 -6213.664,E2 -6213.664} C_VEL
LIN {X 0,Y 495.039,Z 473.088,A -85,B 0,C 180,E1 -6214.48,E2 -6214.48} C_VEL
LIN {X 0,Y 495.143,Z 469.688,A -85,B 0,C 180,E1 -6215.295,E2 -6215.295} C_VEL
LIN {X 0,Y 495.202,Z 465.557,A -85,B 0,C 180,E1 -6216.112,E2 -6216.112} C_VEL
LIN {X 0,Y 495.364,Z 459.279,A -85,B 0,C 180,E1 -6217.112,E2 -6217.112} C_VEL
LIN {X 0,Y 495.43,Z 452.837,A -85,B 0,C 180,E1 -6217.951,E2 -6217.951} C_VEL
LIN {X 0,Y 495.622,Z 446.22,A -85,B 0,C 180,E1 -6218.667,E2 -6218.667} C_VEL
LIN {X 0,Y 495.878,Z 438.209,A -85,B 0,C 180,E1 -6219.382,E2 -6219.382} C_VEL
LIN {X 0,Y 496.073,Z 428.215,A -85,B 0,C 180,E1 -6220.099,E2 -6220.099} C_VEL
LIN {X 0,Y 496.364,Z 416.498,A -85,B 0,C 180,E1 -6220.711,E2 -6220.711} C_VEL
LIN {X 0,Y 496.471,Z 407.043,A -85,B 0,C 180,E1 -6221.07,E2 -6221.07} C_VEL
LIN {X 0,Y 496.666,Z 398.39,A -85,B 0,C 180,E1 -6221.298,E2 -6221.298} C_VEL
LIN {X 0,Y 496.963,Z 331.642,A -85,B 0,C 180,E1 -6222.374,E2 -6222.374} C_VEL
LIN {X 0,Y 495.537,Z 319.954,A -85,B 0,C 180,E1 -6222.605,E2 -6222.605} C_VEL
LIN {X 0,Y 495.791,Z 302.474,A -85,B 0,C 180,E1 -6225.626,E2 -6225.626} C_VEL
LIN {X 0,Y 495.979,Z 286.81,A -85,B 0,C 180,E1 -6228.304,E2 -6228.304} C_VEL
LIN {X 0,Y 496.174,Z 269.932,A -85,B 0,C 180,E1 -6231.174,E2 -6231.174} C_VEL
LIN {X 0,Y 495.843,Z 263.74,A -85,B 0,C 180,E1 -6232.227,E2 -6232.227} C_VEL
LIN {X 0,Y 495.723,Z 263.551,A -85,B 0,C 180,E1 -6235.172,E2 -6235.172} C_VEL
LIN {X 0,Y 495.718,Z 263.549,A -85,B 0,C 180,E1 -6237.896,E2 -6237.896} C_VEL
LIN {X 0,Y 495.717,Z 263.553,A -85,B 0,C 180,E1 -6240.691,E2 -6240.691} C_VEL
LIN {X 0,Y 495.699,Z 263.549,A -85,B 0,C 180,E1 -6243.57,E2 -6243.57} C_VEL
LIN {X 0,Y 495.648,Z 263.558,A -85,B 0,C 180,E1 -6246.552,E2 -6246.552} C_VEL
LIN {X 0,Y 495.721,Z 263.544,A -85,B 0,C 180,E1 -6249.642,E2 -6249.642} C_VEL
LIN {X 0,Y 495.703,Z 263.554,A -85,B 0,C 180,E1 -6252.887,E2 -6252.887} C_VEL
LIN {X 0,Y 495.727,Z 263.542,A -85,B 0,C 180,E1 -6255.996,E2 -6255.996} C_VEL
LIN {X 0,Y 495.74,Z 263.544,A -85,B 0,C 180,E1 -6259.295,E2 -6259.295} C_VEL
LIN {X 0,Y 495.726,Z 263.543,A -85,B 0,C 180,E1 -6262.435,E2 -6262.435} C_VEL
LIN {X 0,Y 495.78,Z 263.54,A -85,B 0,C 180,E1 -6265.454,E2 -6265.454} C_VEL
LIN {X 0,Y 495.768,Z 263.54,A -85,B 0,C 180,E1 -6268.362,E2 -6268.362} C_VEL
LIN {X 0,Y 495.755,Z 263.544,A -85,B 0,C 180,E1 -6271.515,E2 -6271.515} C_VEL
LIN {X 0,Y 495.749,Z 263.544,A -85,B 0,C 180,E1 -6273.927,E2 -6273.927} C_VEL
LIN {X 0,Y 495.773,Z 263.547,A -85,B 0,C 180,E1 -6277.138,E2 -6277.138} C_VEL
LIN {X 0,Y 495.784,Z 263.538,A -85,B 0,C 180,E1 -6280.107,E2 -6280.107} C_VEL
LIN {X 0,Y 495.915,Z 263.529,A -85,B 0,C 180,E1 -6283.531,E2 -6283.531} C_VEL
LIN {X 0,Y 495.86,Z 263.611,A -85,B 0,C 180,E1 -6284.46,E2 -6284.46} C_VEL
LIN {X 0,Y 495.543,Z 281.976,A -85,B 0,C 180,E1 -6287.089,E2 -6287.089} C_VEL
LIN {X 0,Y 495.591,Z 284.527,A -85,B 0,C 180,E1 -6287.436,E2 -6287.436} C_VEL
LIN {X 0,Y 497.238,Z 297.298,A -85,B 0,C 180,E1 -6287.694,E2 -6287.694} C_VEL
LIN {X 0,Y 496.736,Z 362.797,A -85,B 0,C 180,E1 -6288.753,E2 -6288.753} C_VEL
LIN {X 0,Y 496.587,Z 373.077,A -85,B 0,C 180,E1 -6289.033,E2 -6289.033} C_VEL
LIN {X 0,Y 496.392,Z 384.274,A -85,B 0,C 180,E1 -6289.493,E2 -6289.493} C_VEL
LIN {X 0,Y 496.244,Z 393.268,A -85,B 0,C 180,E1 -6290.006,E2 -6290.006} C_VEL
LIN {X 0,Y 496.073,Z 401.796,A -85,B 0,C 180,E1 -6290.62,E2 -6290.62} C_VEL
LIN {X 0,Y 495.885,Z 409.833,A -85,B 0,C 180,E1 -6291.336,E2 -6291.336} C_VEL
LIN {X 0,Y 495.678,Z 416.462,A -85,B 0,C 180,E1 -6292.05,E2 -6292.05} C_VEL
LIN {X 0,Y 495.486,Z 422.633,A -85,B 0,C 180,E1 -6292.851,E2 -6292.851} C_VEL
LIN {X 0,Y 495.451,Z 429.134,A -85,B 0,C 180,E1 -6293.889,E2 -6293.889} C_VEL
LIN {X 0,Y 495.142,Z 435.113,A -85,B 0,C 180,E1 -6295.111,E2 -6295.111} C_VEL
LIN {X 0,Y 495.154,Z 439.391,A -85,B 0,C 180,E1 -6296.334,E2 -6296.334} C_VEL
LIN {X 0,Y 495.07,Z 442.379,A -85,B 0,C 180,E1 -6297.555,E2 -6297.555} C_VEL
LIN {X 0,Y 494.966,Z 443.699,A -85,B 0,C 180,E1 -6298.369,E2 -6298.369} C_VEL
LIN {X 0,Y 494.915,Z 444.53,A -85,B 0,C 180,E1 -6299.182,E2 -6299.182} C_VEL
LIN {X 0,Y 494.906,Z 444.83,A -85,B 0,C 180,E1 -6299.996,E2 -6299.996} C_VEL
LIN {X 0,Y 494.916,Z 444.541,A -85,B 0,C 180,E1 -6300.81,E2 -6300.81} C_VEL
LIN {X 0,Y 494.964,Z 443.767,A -85,B 0,C 180,E1 -6301.623,E2 -6301.623} C_VEL
LIN {X 0,Y 495.069,Z 442.506,A -85,B 0,C 180,E1 -6302.437,E2 -6302.437} C_VEL
LIN {X 0,Y 495.143,Z 439.566,A -85,B 0,C 180,E1 -6303.658,E2 -6303.658} C_VEL
LIN {X 0,Y 495.19,Z 436.886,A -85,B 0,C 180,E1 -6304.473,E2 -6304.473} C_VEL
LIN {X 0,Y 495.166,Z 433.58,A -85,B 0,C 180,E1 -6305.289,E2 -6305.289} C_VEL
LIN {X 0,Y 495.5,Z 428.365,A -85,B 0,C 180,E1 -6306.306,E2 -6306.306} C_VEL
LIN {X 0,Y 495.455,Z 423.673,A -85,B 0,C 180,E1 -6307.067,E2 -6307.067} C_VEL
LIN {X 0,Y 495.632,Z 417.102,A -85,B 0,C 180,E1 -6307.942,E2 -6307.942} C_VEL
LIN {X 0,Y 495.822,Z 410.63,A -85,B 0,C 180,E1 -6308.657,E2 -6308.657} C_VEL
LIN {X 0,Y 496.018,Z 402.798,A -85,B 0,C 180,E1 -6309.373,E2 -6309.373} C_VEL
LIN {X 0,Y 496.207,Z 394.543,A -85,B 0,C 180,E1 -6309.987,E2 -6309.987} C_VEL
LIN {X 0,Y 496.429,Z 384.061,A -85,B 0,C 180,E1 -6310.601,E2 -6310.601} C_VEL
LIN {X 0,Y 496.671,Z 372.146,A -85,B 0,C 180,E1 -6311.085,E2 -6311.085} C_VEL
LIN {X 0,Y 496.772,Z 362.801,A -85,B 0,C 180,E1 -6311.341,E2 -6311.341} C_VEL
LIN {X 0,Y 497.022,Z 294.85,A -85,B 0,C 180,E1 -6312.428,E2 -6312.428} C_VEL
LIN {X 0,Y 495.616,Z 286.202,A -85,B 0,C 180,E1 -6312.619,E2 -6312.619} C_VEL
LIN {X 0,Y 495.814,Z 273.687,A -85,B 0,C 180,E1 -6315.619,E2 -6315.619} C_VEL
LIN {X 0,Y 495.937,Z 264.195,A -85,B 0,C 180,E1 -6317.947,E2 -6317.947} C_VEL
LIN {X 0,Y 495.827,Z 263.536,A -85,B 0,C 180,E1 -6318.164,E2 -6318.164} C_VEL
LIN {X 0,Y 495.727,Z 263.546,A -85,B 0,C 180,E1 -6321.624,E2 -6321.624} C_VEL
LIN {X 0,Y 495.696,Z 263.548,A -85,B 0,C 180,E1 -6324.272,E2 -6324.272} C_VEL
LIN {X 0,Y 495.713,Z 263.551,A -85,B 0,C 180,E1 -6326.974,E2 -6326.974} C_VEL
LIN {X 0,Y 495.736,Z 263.543,A -85,B 0,C 180,E1 -6330.14,E2 -6330.14} C_VEL
LIN {X 0,Y 495.769,Z 263.544,A -85,B 0,C 180,E1 -6333.239,E2 -6333.239} C_VEL
LIN {X 0,Y 495.685,Z 263.551,A -85,B 0,C 180,E1 -6336.082,E2 -6336.082} C_VEL
LIN {X 0,Y 495.732,Z 263.544,A -85,B 0,C 180,E1 -6338.762,E2 -6338.762} C_VEL
LIN {X 0,Y 495.718,Z 263.55,A -85,B 0,C 180,E1 -6341.777,E2 -6341.777} C_VEL
LIN {X 0,Y 495.702,Z 263.549,A -85,B 0,C 180,E1 -6345.136,E2 -6345.136} C_VEL
LIN {X 0,Y 495.709,Z 263.549,A -85,B 0,C 180,E1 -6348.054,E2 -6348.054} C_VEL
LIN {X 0,Y 495.068,Z 263.63,A -85,B 0,C 180,E1 -6348.731,E2 -6348.731} C_VEL
LIN {X 0,Y 492.199,Z 263.988,A -85,B 0,C 180,E1 -6349.831,E2 -6349.831} C_VEL
LIN {X 0,Y 489.758,Z 264.289,A -85,B 0,C 180,E1 -6350.717,E2 -6350.717} C_VEL
LIN {X 0,Y 488.716,Z 264.421,A -85,B 0,C 180,E1 -6351.402,E2 -6351.402} C_VEL
LIN {X 0,Y 488.635,Z 264.431,A -85,B 0,C 180,E1 -6351.633,E2 -6351.633} C_VEL
LIN {X 0,Y 488.684,Z 264.422,A -85,B 0,C 180,E1 -6355.047,E2 -6355.047} C_VEL
LIN {X 0,Y 488.658,Z 264.429,A -85,B 0,C 180,E1 -6358.041,E2 -6358.041} C_VEL
LIN {X 0,Y 488.677,Z 264.424,A -85,B 0,C 180,E1 -6360.726,E2 -6360.726} C_VEL
LIN {X 0,Y 488.718,Z 264.419,A -85,B 0,C 180,E1 -6363.525,E2 -6363.525} C_VEL
LIN {X 0,Y 488.642,Z 264.431,A -85,B 0,C 180,E1 -6366.251,E2 -6366.251} C_VEL
LIN {X 0,Y 488.693,Z 264.421,A -85,B 0,C 180,E1 -6369.172,E2 -6369.172} C_VEL
LIN {X 0,Y 488.678,Z 264.427,A -85,B 0,C 180,E1 -6372.42,E2 -6372.42} C_VEL
LIN {X 0,Y 488.705,Z 264.422,A -85,B 0,C 180,E1 -6374.997,E2 -6374.997} C_VEL
LIN {X 0,Y 488.774,Z 264.416,A -85,B 0,C 180,E1 -6378.386,E2 -6378.386} C_VEL
LIN {X 0,Y 488.76,Z 264.412,A -85,B 0,C 180,E1 -6381.731,E2 -6381.731} C_VEL
LIN {X 0,Y 488.813,Z 264.408,A -85,B 0,C 180,E1 -6384.222,E2 -6384.222} C_VEL
LIN {X 0,Y 488.906,Z 264.395,A -85,B 0,C 180,E1 -6387.527,E2 -6387.527} C_VEL
LIN {X 0,Y 488.905,Z 264.395,A -85,B 0,C 180,E1 -6389.999,E2 -6389.999} C_VEL
LIN {X 0,Y 488.906,Z 264.397,A -85,B 0,C 180,E1 -6392.47,E2 -6392.47} C_VEL
LIN {X 0,Y 488.81,Z 264.407,A -85,B 0,C 180,E1 -6395.775,E2 -6395.775} C_VEL
LIN {X 0,Y 488.764,Z 264.412,A -85,B 0,C 180,E1 -6398.266,E2 -6398.266} C_VEL
LIN {X 0,Y 488.772,Z 264.414,A -85,B 0,C 180,E1 -6401.612,E2 -6401.612} C_VEL
LIN {X 0,Y 488.7,Z 264.425,A -85,B 0,C 180,E1 -6405.001,E2 -6405.001} C_VEL
LIN {X 0,Y 488.693,Z 264.421,A -85,B 0,C 180,E1 -6408.443,E2 -6408.443} C_VEL
LIN {X 0,Y 488.649,Z 264.43,A -85,B 0,C 180,E1 -6411.072,E2 -6411.072} C_VEL
LIN {X 0,Y 488.639,Z 264.432,A -85,B 0,C 180,E1 -6413.746,E2 -6413.746} C_VEL
LIN {X 0,Y 488.739,Z 264.416,A -85,B 0,C 180,E1 -6416.947,E2 -6416.947} C_VEL
LIN {X 0,Y 488.66,Z 264.426,A -85,B 0,C 180,E1 -6420.367,E2 -6420.367} C_VEL
LIN {X 0,Y 488.679,Z 264.427,A -85,B 0,C 180,E1 -6423.487,E2 -6423.487} C_VEL
LIN {X 0,Y 488.633,Z 264.431,A -85,B 0,C 180,E1 -6426.358,E2 -6426.358} C_VEL
LIN {X 0,Y 488.703,Z 264.42,A -85,B 0,C 180,E1 -6429.252,E2 -6429.252} C_VEL
LIN {X 0,Y 488.682,Z 264.425,A -85,B 0,C 180,E1 -6432.524,E2 -6432.524} C_VEL
LIN {X 0,Y 488.661,Z 264.425,A -85,B 0,C 180,E1 -6435.202,E2 -6435.202} C_VEL
LIN {X 0,Y 488.686,Z 264.423,A -85,B 0,C 180,E1 -6437.483,E2 -6437.483} C_VEL
LIN {X 0,Y 488.696,Z 264.423,A -85,B 0,C 180,E1 -6440.753,E2 -6440.753} C_VEL
LIN {X 0,Y 488.641,Z 264.43,A -85,B 0,C 180,E1 -6443.872,E2 -6443.872} C_VEL
LIN {X 0,Y 488.697,Z 264.423,A -85,B 0,C 180,E1 -6446.881,E2 -6446.881} C_VEL
LIN {X 0,Y 488.683,Z 264.423,A -85,B 0,C 180,E1 -6449.785,E2 -6449.785} C_VEL
LIN {X 0,Y 488.693,Z 264.425,A -85,B 0,C 180,E1 -6452.606,E2 -6452.606} C_VEL
LIN {X 0,Y 488.664,Z 264.425,A -85,B 0,C 180,E1 -6455.356,E2 -6455.356} C_VEL
LIN {X 0,Y 488.663,Z 264.425,A -85,B 0,C 180,E1 -6458.047,E2 -6458.047} C_VEL
LIN {X 0,Y 488.707,Z 264.424,A -85,B 0,C 180,E1 -6460.691,E2 -6460.691} C_VEL
LIN {X 0,Y 488.732,Z 264.417,A -85,B 0,C 180,E1 -6464.149,E2 -6464.149} C_VEL
LIN {X 0,Y 488.713,Z 264.42,A -85,B 0,C 180,E1 -6467.548,E2 -6467.548} C_VEL
LIN {X 0,Y 488.73,Z 264.416,A -85,B 0,C 180,E1 -6470.068,E2 -6470.068} C_VEL
LIN {X 0,Y 488.843,Z 264.406,A -85,B 0,C 180,E1 -6472.729,E2 -6472.729} C_VEL
LIN {X 0,Y 488.779,Z 264.415,A -85,B 0,C 180,E1 -6475.055,E2 -6475.055} C_VEL
LIN {X 0,Y 488.928,Z 264.396,A -85,B 0,C 180,E1 -6477.533,E2 -6477.533} C_VEL
LIN {X 0,Y 488.922,Z 264.393,A -85,B 0,C 180,E1 -6480.004,E2 -6480.004} C_VEL
LIN {X 0,Y 488.933,Z 264.391,A -85,B 0,C 180,E1 -6482.476,E2 -6482.476} C_VEL
LIN {X 0,Y 488.812,Z 264.41,A -85,B 0,C 180,E1 -6485.78,E2 -6485.78} C_VEL
LIN {X 0,Y 488.765,Z 264.412,A -85,B 0,C 180,E1 -6488.271,E2 -6488.271} C_VEL
LIN {X 0,Y 488.793,Z 264.413,A -85,B 0,C 180,E1 -6491.616,E2 -6491.616} C_VEL
LIN {X 0,Y 488.739,Z 264.416,A -85,B 0,C 180,E1 -6495.005,E2 -6495.005} C_VEL
LIN {X 0,Y 488.735,Z 264.417,A -85,B 0,C 180,E1 -6498.446,E2 -6498.446} C_VEL
LIN {X 0,Y 488.698,Z 264.42,A -85,B 0,C 180,E1 -6501.074,E2 -6501.074} C_VEL
LIN {X 0,Y 488.662,Z 264.43,A -85,B 0,C 180,E1 -6503.75,E2 -6503.75} C_VEL
LIN {X 0,Y 488.693,Z 264.421,A -85,B 0,C 180,E1 -6506.925,E2 -6506.925} C_VEL
LIN {X 0,Y 488.717,Z 264.422,A -85,B 0,C 180,E1 -6510.223,E2 -6510.223} C_VEL
LIN {X 0,Y 488.705,Z 264.42,A -85,B 0,C 180,E1 -6513.483,E2 -6513.483} C_VEL
LIN {X 0,Y 488.66,Z 264.429,A -85,B 0,C 180,E1 -6516.354,E2 -6516.354} C_VEL
LIN {X 0,Y 488.683,Z 264.422,A -85,B 0,C 180,E1 -6519.259,E2 -6519.259} C_VEL
LIN {X 0,Y 488.664,Z 264.429,A -85,B 0,C 180,E1 -6522.531,E2 -6522.531} C_VEL
LIN {X 0,Y 488.695,Z 264.422,A -85,B 0,C 180,E1 -6525.199,E2 -6525.199} C_VEL
LIN {X 0,Y 488.66,Z 264.429,A -85,B 0,C 180,E1 -6528.582,E2 -6528.582} C_VEL
LIN {X 0,Y 488.688,Z 264.425,A -85,B 0,C 180,E1 -6530.952,E2 -6530.952} C_VEL
LIN {X 0,Y 488.664,Z 264.424,A -85,B 0,C 180,E1 -6533.869,E2 -6533.869} C_VEL
LIN {X 0,Y 488.701,Z 264.424,A -85,B 0,C 180,E1 -6536.877,E2 -6536.877} C_VEL
LIN {X 0,Y 488.705,Z 264.419,A -85,B 0,C 180,E1 -6539.782,E2 -6539.782} C_VEL
LIN {X 0,Y 488.697,Z 264.424,A -85,B 0,C 180,E1 -6543.081,E2 -6543.081} C_VEL
LIN {X 0,Y 488.762,Z 264.622,A -85,B 0,C 180,E1 -6546.306,E2 -6546.306} C_VEL
LIN {X 0,Y 489.976,Z 272.272,A -85,B 0,C 180,E1 -6547.884,E2 -6547.884} C_VEL
LIN {X 0,Y 489.504,Z 287.866,A -85,B 0,C 180,E1 -6550.923,E2 -6550.923} C_VEL
LIN {X 0,Y 488.95,Z 305.84,A -85,B 0,C 180,E1 -6554.377,E2 -6554.377} C_VEL
LIN {X 0,Y 488.567,Z 320.86,A -85,B 0,C 180,E1 -6557.227,E2 -6557.227} C_VEL
LIN {X 0,Y 490.182,Z 334.88,A -85,B 0,C 180,E1 -6557.503,E2 -6557.503} C_VEL
LIN {X 0,Y 489.723,Z 398.553,A -85,B 0,C 180,E1 -6558.542,E2 -6558.542} C_VEL
LIN {X 0,Y 489.522,Z 408.8,A -85,B 0,C 180,E1 -6558.826,E2 -6558.826} C_VEL
LIN {X 0,Y 489.255,Z 420.944,A -85,B 0,C 180,E1 -6559.344,E2 -6559.344} C_VEL
LIN {X 0,Y 489.029,Z 429.776,A -85,B 0,C 180,E1 -6559.862,E2 -6559.862} C_VEL
LIN {X 0,Y 488.856,Z 438.212,A -85,B 0,C 180,E1 -6560.485,E2 -6560.485} C_VEL
LIN {X 0,Y 488.608,Z 446.189,A -85,B 0,C 180,E1 -6561.211,E2 -6561.211} C_VEL
LIN {X 0,Y 488.411,Z 452.785,A -85,B 0,C 180,E1 -6561.936,E2 -6561.936} C_VEL
LIN {X 0,Y 488.285,Z 459.061,A -85,B 0,C 180,E1 -6562.766,E2 -6562.766} C_VEL
LIN {X 0,Y 488.115,Z 464.871,A -85,B 0,C 180,E1 -6563.701,E2 -6563.701} C_VEL
LIN {X 0,Y 488.077,Z 469.562,A -85,B 0,C 180,E1 -6564.631,E2 -6564.631} C_VEL
LIN {X 0,Y 487.948,Z 474.468,A -85,B 0,C 180,E1 -6565.872,E2 -6565.872} C_VEL
LIN {X 0,Y 487.987,Z 476.857,A -85,B 0,C 180,E1 -6566.699,E2 -6566.699} C_VEL
LIN {X 0,Y 487.914,Z 478.669,A -85,B 0,C 180,E1 -6567.525,E2 -6567.525} C_VEL
LIN {X 0,Y 487.892,Z 479.965,A -85,B 0,C 180,E1 -6568.351,E2 -6568.351} C_VEL
LIN {X 0,Y 487.835,Z 480.764,A -85,B 0,C 180,E1 -6569.176,E2 -6569.176} C_VEL
LIN {X 0,Y 487.823,Z 481.053,A -85,B 0,C 180,E1 -6570.001,E2 -6570.001} C_VEL
LIN {X 0,Y 487.835,Z 480.737,A -85,B 0,C 180,E1 -6570.827,E2 -6570.827} C_VEL
LIN {X 0,Y 487.892,Z 479.915,A -85,B 0,C 180,E1 -6571.652,E2 -6571.652} C_VEL
LIN {X 0,Y 487.914,Z 478.596,A -85,B 0,C 180,E1 -6572.478,E2 -6572.478} C_VEL
LIN {X 0,Y 488.007,Z 475.571,A -85,B 0,C 180,E1 -6573.717,E2 -6573.717} C_VEL
LIN {X 0,Y 487.951,Z 472.798,A -85,B 0,C 180,E1 -6574.545,E2 -6574.545} C_VEL
LIN {X 0,Y 488.078,Z 469.388,A -85,B 0,C 180,E1 -6575.372,E2 -6575.372} C_VEL
LIN {X 0,Y 488.105,Z 464.733,A -85,B 0,C 180,E1 -6576.288,E2 -6576.288} C_VEL
LIN {X 0,Y 488.289,Z 458.797,A -85,B 0,C 180,E1 -6577.236,E2 -6577.236} C_VEL
LIN {X 0,Y 488.375,Z 452.476,A -85,B 0,C 180,E1 -6578.067,E2 -6578.067} C_VEL
LIN {X 0,Y 488.603,Z 445.831,A -85,B 0,C 180,E1 -6578.792,E2 -6578.792} C_VEL
LIN {X 0,Y 488.861,Z 437.78,A -85,B 0,C 180,E1 -6579.518,E2 -6579.518} C_VEL
LIN {X 0,Y 489.065,Z 427.742,A -85,B 0,C 180,E1 -6580.245,E2 -6580.245} C_VEL
LIN {X 0,Y 489.358,Z 417.133,A -85,B 0,C 180,E1 -6580.814,E2 -6580.814} C_VEL
LIN {X 0,Y 489.472,Z 407.202,A -85,B 0,C 180,E1 -6581.204,E2 -6581.204} C_VEL
LIN {X 0,Y 489.694,Z 397.575,A -85,B 0,C 180,E1 -6581.461,E2 -6581.461} C_VEL
LIN {X 0,Y 490.076,Z 332.591,A -85,B 0,C 180,E1 -6582.537,E2 -6582.537} C_VEL
LIN {X 0,Y 488.52,Z 319.65,A -85,B 0,C 180,E1 -6582.804,E2 -6582.804} C_VEL
LIN {X 0,Y 488.796,Z 300.919,A -85,B 0,C 180,E1 -6586.069,E2 -6586.069} C_VEL
LIN {X 0,Y 489.038,Z 282.136,A -85,B 0,C 180,E1 -6589.302,E2 -6589.302} C_VEL
LIN {X 0,Y 489.178,Z 268.02,A -85,B 0,C 180,E1 -6591.714,E2 -6591.714} C_VEL
LIN {X 0,Y 488.755,Z 264.42,A -85,B 0,C 180,E1 -6592.344,E2 -6592.344} C_VEL
LIN {X 0,Y 488.659,Z 264.428,A -85,B 0,C 180,E1 -6595.562,E2 -6595.562} C_VEL
LIN {X 0,Y 488.694,Z 264.426,A -85,B 0,C 180,E1 -6598.333,E2 -6598.333} C_VEL
LIN {X 0,Y 488.663,Z 264.429,A -85,B 0,C 180,E1 -6601.183,E2 -6601.183} C_VEL
LIN {X 0,Y 488.644,Z 264.427,A -85,B 0,C 180,E1 -6604.121,E2 -6604.121} C_VEL
LIN {X 0,Y 488.64,Z 264.432,A -85,B 0,C 180,E1 -6607.164,E2 -6607.164} C_VEL
LIN {X 0,Y 488.68,Z 264.424,A -85,B 0,C 180,E1 -6609.257,E2 -6609.257} C_VEL
LIN {X 0,Y 488.661,Z 264.426,A -85,B 0,C 180,E1 -6612.53,E2 -6612.53} C_VEL
LIN {X 0,Y 488.71,Z 264.422,A -85,B 0,C 180,E1 -6615.196,E2 -6615.196} C_VEL
LIN {X 0,Y 488.675,Z 264.423,A -85,B 0,C 180,E1 -6618.578,E2 -6618.578} C_VEL
LIN {X 0,Y 488.703,Z 264.424,A -85,B 0,C 180,E1 -6620.949,E2 -6620.949} C_VEL
LIN {X 0,Y 488.679,Z 264.42,A -85,B 0,C 180,E1 -6623.865,E2 -6623.865} C_VEL
LIN {X 0,Y 488.717,Z 264.423,A -85,B 0,C 180,E1 -6626.873,E2 -6626.873} C_VEL
LIN {X 0,Y 488.734,Z 264.417,A -85,B 0,C 180,E1 -6629.779,E2 -6629.779} C_VEL
LIN {X 0,Y 488.728,Z 264.424,A -85,B 0,C 180,E1 -6633.073,E2 -6633.073} C_VEL
LIN {X 0,Y 488.687,Z 264.424,A -85,B 0,C 180,E1 -6636.251,E2 -6636.251} C_VEL
LIN {X 0,Y 488.761,Z 264.419,A -85,B 0,C 180,E1 -6639.173,E2 -6639.173} C_VEL
LIN {X 0,Y 488.772,Z 264.414,A -85,B 0,C 180,E1 -6642.422,E2 -6642.422} C_VEL
LIN {X 0,Y 488.871,Z 264.51,A -85,B 0,C 180,E1 -6644.376,E2 -6644.376} C_VEL
LIN {X 0,Y 488.564,Z 282.227,A -85,B 0,C 180,E1 -6646.901,E2 -6646.901} C_VEL
LIN {X 0,Y 488.557,Z 284.236,A -85,B 0,C 180,E1 -6647.209,E2 -6647.209} C_VEL
LIN {X 0,Y 490.352,Z 298.394,A -85,B 0,C 180,E1 -6647.518,E2 -6647.518} C_VEL
LIN {X 0,Y 489.77,Z 363.802,A -85,B 0,C 180,E1 -6648.617,E2 -6648.617} C_VEL
LIN {X 0,Y 489.629,Z 374.625,A -85,B 0,C 180,E1 -6648.928,E2 -6648.928} C_VEL
LIN {X 0,Y 489.392,Z 386.225,A -85,B 0,C 180,E1 -6649.446,E2 -6649.446} C_VEL
LIN {X 0,Y 489.19,Z 394.886,A -85,B 0,C 180,E1 -6649.965,E2 -6649.965} C_VEL
LIN {X 0,Y 489.051,Z 403.179,A -85,B 0,C 180,E1 -6650.588,E2 -6650.588} C_VEL
LIN {X 0,Y 488.832,Z 411.039,A -85,B 0,C 180,E1 -6651.314,E2 -6651.314} C_VEL
LIN {X 0,Y 488.613,Z 418.379,A -85,B 0,C 180,E1 -6652.143,E2 -6652.143} C_VEL
LIN {X 0,Y 488.416,Z 425.661,A -85,B 0,C 180,E1 -6653.157,E2 -6653.157} C_VEL
LIN {X 0,Y 488.26,Z 431.576,A -85,B 0,C 180,E1 -6654.213,E2 -6654.213} C_VEL
LIN {X 0,Y 488.065,Z 435.371,A -85,B 0,C 180,E1 -6655.04,E2 -6655.04} C_VEL
LIN {X 0,Y 488.138,Z 438.428,A -85,B 0,C 180,E1 -6655.868,E2 -6655.868} C_VEL
LIN {X 0,Y 488.051,Z 440.818,A -85,B 0,C 180,E1 -6656.694,E2 -6656.694} C_VEL
LIN {X 0,Y 488.007,Z 442.649,A -85,B 0,C 180,E1 -6657.52,E2 -6657.52} C_VEL
LIN {X 0,Y 487.896,Z 443.97,A -85,B 0,C 180,E1 -6658.345,E2 -6658.345} C_VEL
LIN {X 0,Y 487.838,Z 444.798,A -85,B 0,C 180,E1 -6659.17,E2 -6659.17} C_VEL
LIN {X 0,Y 487.827,Z 445.095,A -85,B 0,C 180,E1 -6659.996,E2 -6659.996} C_VEL
LIN {X 0,Y 487.839,Z 444.8,A -85,B 0,C 180,E1 -6660.821,E2 -6660.821} C_VEL
LIN {X 0,Y 487.894,Z 444.016,A -85,B 0,C 180,E1 -6661.647,E2 -6661.647} C_VEL
LIN {X 0,Y 487.977,Z 442.74,A -85,B 0,C 180,E1 -6662.472,E2 -6662.472} C_VEL
LIN {X 0,Y 488.071,Z 439.78,A -85,B 0,C 180,E1 -6663.711,E2 -6663.711} C_VEL
LIN {X 0,Y 488.102,Z 437.078,A -85,B 0,C 180,E1 -6664.538,E2 -6664.538} C_VEL
LIN {X 0,Y 488.112,Z 433.744,A -85,B 0,C 180,E1 -6665.366,E2 -6665.366} C_VEL
LIN {X 0,Y 488.448,Z 428.499,A -85,B 0,C 180,E1 -6666.398,E2 -6666.398} C_VEL
LIN {X 0,Y 488.44,Z 422.965,A -85,B 0,C 180,E1 -6667.285,E2 -6667.285} C_VEL
LIN {X 0,Y 488.652,Z 415.434,A -85,B 0,C 180,E1 -6668.265,E2 -6668.265} C_VEL
LIN {X 0,Y 488.932,Z 406.444,A -85,B 0,C 180,E1 -6669.197,E2 -6669.197} C_VEL
LIN {X 0,Y 489.142,Z 397.437,A -85,B 0,C 180,E1 -6669.924,E2 -6669.924} C_VEL
LIN {X 0,Y 489.367,Z 389.475,A -85,B 0,C 180,E1 -6670.441,E2 -6670.441} C_VEL
LIN {X 0,Y 489.526,Z 380.345,A -85,B 0,C 180,E1 -6670.909,E2 -6670.909} C_VEL
LIN {X 0,Y 489.683,Z 370.798,A -85,B 0,C 180,E1 -6671.272,E2 -6671.272} C_VEL
LIN {X 0,Y 489.785,Z 361.891,A -85,B 0,C 180,E1 -6671.505,E2 -6671.505} C_VEL
LIN {X 0,Y 490.122,Z 295.905,A -85,B 0,C 180,E1 -6672.585,E2 -6672.585} C_VEL
LIN {X 0,Y 488.563,Z 286.383,A -85,B 0,C 180,E1 -6672.805,E2 -6672.805} C_VEL
LIN {X 0,Y 488.798,Z 273.811,A -85,B 0,C 180,E1 -6675.849,E2 -6675.849} C_VEL
LIN {X 0,Y 488.924,Z 265.199,A -85,B 0,C 180,E1 -6677.983,E2 -6677.983} C_VEL
LIN {X 0,Y 488.793,Z 264.413,A -85,B 0,C 180,E1 -6678.195,E2 -6678.195} C_VEL
LIN {X 0,Y 488.695,Z 264.425,A -85,B 0,C 180,E1 -6681.066,E2 -6681.066} C_VEL
LIN {X 0,Y 488.653,Z 264.427,A -85,B 0,C 180,E1 -6683.742,E2 -6683.742} C_VEL
LIN {X 0,Y 488.68,Z 264.428,A -85,B 0,C 180,E1 -6686.916,E2 -6686.916} C_VEL
LIN {X 0,Y 488.695,Z 264.421,A -85,B 0,C 180,E1 -6690.215,E2 -6690.215} C_VEL
LIN {X 0,Y 488.711,Z 264.423,A -85,B 0,C 180,E1 -6693.479,E2 -6693.479} C_VEL
LIN {X 0,Y 488.646,Z 264.427,A -85,B 0,C 180,E1 -6696.347,E2 -6696.347} C_VEL
LIN {X 0,Y 488.669,Z 264.429,A -85,B 0,C 180,E1 -6699.249,E2 -6699.249} C_VEL
LIN {X 0,Y 488.664,Z 264.429,A -85,B 0,C 180,E1 -6701.593,E2 -6701.593} C_VEL
LIN {X 0,Y 488.667,Z 264.424,A -85,B 0,C 180,E1 -6704.798,E2 -6704.798} C_VEL
LIN {X 0,Y 488.65,Z 264.427,A -85,B 0,C 180,E1 -6708.057,E2 -6708.057} C_VEL
LIN {X 0,Y 488.663,Z 264.425,A -85,B 0,C 180,E1 -6710.943,E2 -6710.943} C_VEL
LIN {X 0,Y 488.635,Z 264.431,A -85,B 0,C 180,E1 -6711.633,E2 -6711.633} C_VEL
LIN {X 0,Y 487.976,Z 264.517,A -85,B 0,C 180,E1 -6712.321,E2 -6712.321} C_VEL
LIN {X 0,Y 485.114,Z 264.871,A -85,B 0,C 180,E1 -6713.437,E2 -6713.437} C_VEL
LIN {X 0,Y 482.711,Z 265.169,A -85,B 0,C 180,E1 -6714.337,E2 -6714.337} C_VEL
LIN {X 0,Y 481.709,Z 265.291,A -85,B 0,C 180,E1 -6715.032,E2 -6715.032} C_VEL
LIN {X 0,Y 481.645,Z 265.3,A -85,B 0,C 180,E1 -6715.268,E2 -6715.268} C_VEL
LIN {X 0,Y 481.6,Z 265.309,A -85,B 0,C 180,E1 -6718.307,E2 -6718.307} C_VEL
LIN {X 0,Y 481.653,Z 265.298,A -85,B 0,C 180,E1 -6721.214,E2 -6721.214} C_VEL
LIN {X 0,Y 481.658,Z 265.302,A -85,B 0,C 180,E1 -6724.039,E2 -6724.039} C_VEL
LIN {X 0,Y 481.623,Z 265.304,A -85,B 0,C 180,E1 -6726.808,E2 -6726.808} C_VEL
LIN {X 0,Y 481.642,Z 265.3,A -85,B 0,C 180,E1 -6729.499,E2 -6729.499} C_VEL
LIN {X 0,Y 481.652,Z 265.303,A -85,B 0,C 180,E1 -6732.155,E2 -6732.155} C_VEL
LIN {X 0,Y 481.686,Z 265.298,A -85,B 0,C 180,E1 -6734.773,E2 -6734.773} C_VEL
LIN {X 0,Y 481.739,Z 265.291,A -85,B 0,C 180,E1 -6738.214,E2 -6738.214} C_VEL
LIN {X 0,Y 481.706,Z 265.291,A -85,B 0,C 180,E1 -6741.609,E2 -6741.609} C_VEL
LIN {X 0,Y 481.771,Z 265.285,A -85,B 0,C 180,E1 -6744.138,E2 -6744.138} C_VEL
LIN {X 0,Y 481.874,Z 265.271,A -85,B 0,C 180,E1 -6747.491,E2 -6747.491} C_VEL
LIN {X 0,Y 481.876,Z 265.27,A -85,B 0,C 180,E1 -6749.999,E2 -6749.999} C_VEL
LIN {X 0,Y 481.874,Z 265.273,A -85,B 0,C 180,E1 -6752.506,E2 -6752.506} C_VEL
LIN {X 0,Y 481.768,Z 265.284,A -85,B 0,C 180,E1 -6755.859,E2 -6755.859} C_VEL
LIN {X 0,Y 481.71,Z 265.292,A -85,B 0,C 180,E1 -6758.388,E2 -6758.388} C_VEL
LIN {X 0,Y 481.736,Z 265.289,A -85,B 0,C 180,E1 -6761.784,E2 -6761.784} C_VEL
LIN {X 0,Y 481.68,Z 265.299,A -85,B 0,C 180,E1 -6765.225,E2 -6765.225} C_VEL
LIN {X 0,Y 481.651,Z 265.299,A -85,B 0,C 180,E1 -6768.722,E2 -6768.722} C_VEL
LIN {X 0,Y 481.59,Z 265.31,A -85,B 0,C 180,E1 -6771.395,E2 -6771.395} C_VEL
LIN {X 0,Y 481.621,Z 265.304,A -85,B 0,C 180,E1 -6774.114,E2 -6774.114} C_VEL
LIN {X 0,Y 481.693,Z 265.296,A -85,B 0,C 180,E1 -6777.142,E2 -6777.142} C_VEL
LIN {X 0,Y 481.629,Z 265.305,A -85,B 0,C 180,E1 -6779.742,E2 -6779.742} C_VEL
LIN {X 0,Y 481.616,Z 265.303,A -85,B 0,C 180,E1 -6782.676,E2 -6782.676} C_VEL
LIN {X 0,Y 481.587,Z 265.311,A -85,B 0,C 180,E1 -6785.711,E2 -6785.711} C_VEL
LIN {X 0,Y 481.674,Z 265.297,A -85,B 0,C 180,E1 -6789.359,E2 -6789.359} C_VEL
LIN {X 0,Y 481.624,Z 265.305,A -85,B 0,C 180,E1 -6792.161,E2 -6792.161} C_VEL
LIN {X 0,Y 481.61,Z 265.307,A -85,B 0,C 180,E1 -6794.46,E2 -6794.46} C_VEL
LIN {X 0,Y 481.64,Z 265.3,A -85,B 0,C 180,E1 -6796.849,E2 -6796.849} C_VEL
LIN {X 0,Y 481.642,Z 265.304,A -85,B 0,C 180,E1 -6800.064,E2 -6800.064} C_VEL
LIN {X 0,Y 481.584,Z 265.307,A -85,B 0,C 180,E1 -6803.257,E2 -6803.257} C_VEL
LIN {X 0,Y 481.668,Z 265.3,A -85,B 0,C 180,E1 -6806.334,E2 -6806.334} C_VEL
LIN {X 0,Y 481.61,Z 265.303,A -85,B 0,C 180,E1 -6809.422,E2 -6809.422} C_VEL
LIN {X 0,Y 481.654,Z 265.301,A -85,B 0,C 180,E1 -6812.172,E2 -6812.172} C_VEL
LIN {X 0,Y 481.642,Z 265.303,A -85,B 0,C 180,E1 -6814.972,E2 -6814.972} C_VEL
LIN {X 0,Y 481.613,Z 265.303,A -85,B 0,C 180,E1 -6817.709,E2 -6817.709} C_VEL
LIN {X 0,Y 481.67,Z 265.299,A -85,B 0,C 180,E1 -6820.397,E2 -6820.397} C_VEL
LIN {X 0,Y 481.646,Z 265.302,A -85,B 0,C 180,E1 -6823.038,E2 -6823.038} C_VEL
LIN {X 0,Y 481.657,Z 265.298,A -85,B 0,C 180,E1 -6825.643,E2 -6825.643} C_VEL
LIN {X 0,Y 481.724,Z 265.289,A -85,B 0,C 180,E1 -6828.219,E2 -6828.219} C_VEL
LIN {X 0,Y 481.714,Z 265.292,A -85,B 0,C 180,E1 -6831.616,E2 -6831.616} C_VEL
LIN {X 0,Y 481.776,Z 265.283,A -85,B 0,C 180,E1 -6834.144,E2 -6834.144} C_VEL
LIN {X 0,Y 481.895,Z 265.271,A -85,B 0,C 180,E1 -6837.497,E2 -6837.497} C_VEL
LIN {X 0,Y 481.892,Z 265.269,A -85,B 0,C 180,E1 -6840.004,E2 -6840.004} C_VEL
LIN {X 0,Y 481.899,Z 265.267,A -85,B 0,C 180,E1 -6842.512,E2 -6842.512} C_VEL
LIN {X 0,Y 481.771,Z 265.287,A -85,B 0,C 180,E1 -6845.865,E2 -6845.865} C_VEL
LIN {X 0,Y 481.721,Z 265.29,A -85,B 0,C 180,E1 -6848.393,E2 -6848.393} C_VEL
LIN {X 0,Y 481.739,Z 265.291,A -85,B 0,C 180,E1 -6851.789,E2 -6851.789} C_VEL
LIN {X 0,Y 481.72,Z 265.292,A -85,B 0,C 180,E1 -6855.228,E2 -6855.228} C_VEL
LIN {X 0,Y 481.696,Z 265.293,A -85,B 0,C 180,E1 -6858.726,E2 -6858.726} C_VEL
LIN {X 0,Y 481.636,Z 265.302,A -85,B 0,C 180,E1 -6861.398,E2 -6861.398} C_VEL
LIN {X 0,Y 481.641,Z 265.303,A -85,B 0,C 180,E1 -6864.118,E2 -6864.118} C_VEL
LIN {X 0,Y 481.668,Z 265.296,A -85,B 0,C 180,E1 -6867.125,E2 -6867.125} C_VEL
LIN {X 0,Y 481.667,Z 265.3,A -85,B 0,C 180,E1 -6869.745,E2 -6869.745} C_VEL
LIN {X 0,Y 481.647,Z 265.301,A -85,B 0,C 180,E1 -6872.679,E2 -6872.679} C_VEL
LIN {X 0,Y 481.621,Z 265.304,A -85,B 0,C 180,E1 -6875.714,E2 -6875.714} C_VEL
LIN {X 0,Y 481.627,Z 265.303,A -85,B 0,C 180,E1 -6878.866,E2 -6878.866} C_VEL
LIN {X 0,Y 481.622,Z 265.304,A -85,B 0,C 180,E1 -6881.912,E2 -6881.912} C_VEL
LIN {X 0,Y 481.651,Z 265.302,A -85,B 0,C 180,E1 -6884.461,E2 -6884.461} C_VEL
LIN {X 0,Y 481.613,Z 265.303,A -85,B 0,C 180,E1 -6887.838,E2 -6887.838} C_VEL
LIN {X 0,Y 481.648,Z 265.303,A -85,B 0,C 180,E1 -6890.659,E2 -6890.659} C_VEL
LIN {X 0,Y 481.619,Z 265.303,A -85,B 0,C 180,E1 -6893.38,E2 -6893.38} C_VEL
LIN {X 0,Y 481.671,Z 265.298,A -85,B 0,C 180,E1 -6896.329,E2 -6896.329} C_VEL
LIN {X 0,Y 481.635,Z 265.303,A -85,B 0,C 180,E1 -6899.423,E2 -6899.423} C_VEL
LIN {X 0,Y 481.649,Z 265.299,A -85,B 0,C 180,E1 -6902.167,E2 -6902.167} C_VEL
LIN {X 0,Y 481.671,Z 265.303,A -85,B 0,C 180,E1 -6904.969,E2 -6904.969} C_VEL
LIN {X 0,Y 481.695,Z 265.494,A -85,B 0,C 180,E1 -6906.168,E2 -6906.168} C_VEL
LIN {X 0,Y 482.975,Z 273.151,A -85,B 0,C 180,E1 -6907.771,E2 -6907.771} C_VEL
LIN {X 0,Y 482.505,Z 287.798,A -85,B 0,C 180,E1 -6910.672,E2 -6910.672} C_VEL
LIN {X 0,Y 481.955,Z 304.448,A -85,B 0,C 180,E1 -6913.917,E2 -6913.917} C_VEL
LIN {X 0,Y 481.534,Z 320.635,A -85,B 0,C 180,E1 -6917.042,E2 -6917.042} C_VEL
LIN {X 0,Y 483.222,Z 335.741,A -85,B 0,C 180,E1 -6917.353,E2 -6917.353} C_VEL
LIN {X 0,Y 482.732,Z 398.48,A -85,B 0,C 180,E1 -6918.401,E2 -6918.401} C_VEL
LIN {X 0,Y 482.515,Z 409.445,A -85,B 0,C 180,E1 -6918.715,E2 -6918.715} C_VEL
LIN {X 0,Y 482.264,Z 420.271,A -85,B 0,C 180,E1 -6919.187,E2 -6919.187} C_VEL
LIN {X 0,Y 481.972,Z 430.689,A -85,B 0,C 180,E1 -6919.818,E2 -6919.818} C_VEL
LIN {X 0,Y 481.787,Z 438.918,A -85,B 0,C 180,E1 -6920.45,E2 -6920.45} C_VEL
LIN {X 0,Y 481.537,Z 446.739,A -85,B 0,C 180,E1 -6921.186,E2 -6921.186} C_VEL
LIN {X 0,Y 481.264,Z 455.752,A -85,B 0,C 180,E1 -6922.238,E2 -6922.238} C_VEL
LIN {X 0,Y 481.092,Z 462.698,A -85,B 0,C 180,E1 -6923.29,E2 -6923.29} C_VEL
LIN {X 0,Y 481.001,Z 467.27,A -85,B 0,C 180,E1 -6924.131,E2 -6924.131} C_VEL
LIN {X 0,Y 480.933,Z 471.072,A -85,B 0,C 180,E1 -6924.971,E2 -6924.971} C_VEL
LIN {X 0,Y 480.909,Z 475.381,A -85,B 0,C 180,E1 -6926.231,E2 -6926.231} C_VEL
LIN {X 0,Y 480.829,Z 478.383,A -85,B 0,C 180,E1 -6927.488,E2 -6927.488} C_VEL
LIN {X 0,Y 480.823,Z 479.692,A -85,B 0,C 180,E1 -6928.326,E2 -6928.326} C_VEL
LIN {X 0,Y 480.761,Z 480.5,A -85,B 0,C 180,E1 -6929.164,E2 -6929.164} C_VEL
LIN {X 0,Y 480.747,Z 480.79,A -85,B 0,C 180,E1 -6930.001,E2 -6930.001} C_VEL
LIN {X 0,Y 480.761,Z 480.474,A -85,B 0,C 180,E1 -6930.839,E2 -6930.839} C_VEL
LIN {X 0,Y 480.823,Z 479.655,A -85,B 0,C 180,E1 -6931.677,E2 -6931.677} C_VEL
LIN {X 0,Y 480.829,Z 478.332,A -85,B 0,C 180,E1 -6932.515,E2 -6932.515} C_VEL
LIN {X 0,Y 480.91,Z 475.294,A -85,B 0,C 180,E1 -6933.772,E2 -6933.772} C_VEL
LIN {X 0,Y 480.869,Z 472.514,A -85,B 0,C 180,E1 -6934.612,E2 -6934.612} C_VEL
LIN {X 0,Y 480.995,Z 469.09,A -85,B 0,C 180,E1 -6935.451,E2 -6935.451} C_VEL
LIN {X 0,Y 481.056,Z 463.42,A -85,B 0,C 180,E1 -6936.554,E2 -6936.554} C_VEL
LIN {X 0,Y 481.233,Z 456.993,A -85,B 0,C 180,E1 -6937.554,E2 -6937.554} C_VEL
LIN {X 0,Y 481.459,Z 448.544,A -85,B 0,C 180,E1 -6938.606,E2 -6938.606} C_VEL
LIN {X 0,Y 481.748,Z 439.852,A -85,B 0,C 180,E1 -6939.447,E2 -6939.447} C_VEL
LIN {X 0,Y 481.927,Z 431.858,A -85,B 0,C 180,E1 -6940.08,E2 -6940.08} C_VEL
LIN {X 0,Y 482.14,Z 423.677,A -85,B 0,C 180,E1 -6940.606,E2 -6940.606} C_VEL
LIN {X 0,Y 482.409,Z 414.272,A -85,B 0,C 180,E1 -6941.078,E2 -6941.078} C_VEL
LIN {X 0,Y 482.584,Z 405.143,A -85,B 0,C 180,E1 -6941.419,E2 -6941.419} C_VEL
LIN {X 0,Y 482.821,Z 394.717,A -85,B 0,C 180,E1 -6941.68,E2 -6941.68} C_VEL
LIN {X 0,Y 483.138,Z 333,A -85,B 0,C 180,E1 -6942.725,E2 -6942.725} C_VEL
LIN {X 0,Y 481.459,Z 319.208,A -85,B 0,C 180,E1 -6943.019,E2 -6943.019} C_VEL
LIN {X 0,Y 481.742,Z 301.739,A -85,B 0,C 180,E1 -6946.094,E2 -6946.094} C_VEL
LIN {X 0,Y 482.027,Z 284.229,A -85,B 0,C 180,E1 -6949.152,E2 -6949.152} C_VEL
LIN {X 0,Y 482.156,Z 268.823,A -85,B 0,C 180,E1 -6951.821,E2 -6951.821} C_VEL
LIN {X 0,Y 481.714,Z 265.298,A -85,B 0,C 180,E1 -6952.463,E2 -6952.463} C_VEL
LIN {X 0,Y 481.646,Z 265.305,A -85,B 0,C 180,E1 -6955.217,E2 -6955.217} C_VEL
LIN {X 0,Y 481.652,Z 265.302,A -85,B 0,C 180,E1 -6957.836,E2 -6957.836} C_VEL
LIN {X 0,Y 481.618,Z 265.309,A -85,B 0,C 180,E1 -6960.714,E2 -6960.714} C_VEL
LIN {X 0,Y 481.613,Z 265.303,A -85,B 0,C 180,E1 -6963.715,E2 -6963.715} C_VEL
LIN {X 0,Y 481.599,Z 265.309,A -85,B 0,C 180,E1 -6966.75,E2 -6966.75} C_VEL
LIN {X 0,Y 481.642,Z 265.297,A -85,B 0,C 180,E1 -6969.945,E2 -6969.945} C_VEL
LIN {X 0,Y 481.628,Z 265.303,A -85,B 0,C 180,E1 -6973.302,E2 -6973.302} C_VEL
LIN {X 0,Y 481.644,Z 265.298,A -85,B 0,C 180,E1 -6975.644,E2 -6975.644} C_VEL
LIN {X 0,Y 481.637,Z 265.305,A -85,B 0,C 180,E1 -6978.954,E2 -6978.954} C_VEL
LIN {X 0,Y 481.652,Z 265.295,A -85,B 0,C 180,E1 -6981.994,E2 -6981.994} C_VEL
LIN {X 0,Y 481.695,Z 265.295,A -85,B 0,C 180,E1 -6985.316,E2 -6985.316} C_VEL
LIN {X 0,Y 481.657,Z 265.298,A -85,B 0,C 180,E1 -6988.31,E2 -6988.31} C_VEL
LIN {X 0,Y 481.679,Z 265.301,A -85,B 0,C 180,E1 -6991.214,E2 -6991.214} C_VEL
LIN {X 0,Y 481.669,Z 265.298,A -85,B 0,C 180,E1 -6994.038,E2 -6994.038} C_VEL
LIN {X 0,Y 481.689,Z 265.3,A -85,B 0,C 180,E1 -6996.81,E2 -6996.81} C_VEL
LIN {X 0,Y 481.71,Z 265.296,A -85,B 0,C 180,E1 -6999.5,E2 -6999.5} C_VEL
LIN {X 0,Y 481.798,Z 265.287,A -85,B 0,C 180,E1 -7003.034,E2 -7003.034} C_VEL
LIN {X 0,Y 481.892,Z 265.451,A -85,B 0,C 180,E1 -7004.273,E2 -7004.273} C_VEL
LIN {X 0,Y 481.593,Z 284.678,A -85,B 0,C 180,E1 -7007.016,E2 -7007.016} C_VEL
LIN {X 0,Y 483.47,Z 298.472,A -85,B 0,C 180,E1 -7007.317,E2 -7007.317} C_VEL
LIN {X 0,Y 482.83,Z 364.293,A -85,B 0,C 180,E1 -7008.451,E2 -7008.451} C_VEL
LIN {X 0,Y 482.645,Z 376.387,A -85,B 0,C 180,E1 -7008.819,E2 -7008.819} C_VEL
LIN {X 0,Y 482.417,Z 386.507,A -85,B 0,C 180,E1 -7009.292,E2 -7009.292} C_VEL
LIN {X 0,Y 482.216,Z 395.14,A -85,B 0,C 180,E1 -7009.818,E2 -7009.818} C_VEL
LIN {X 0,Y 482.061,Z 403.415,A -85,B 0,C 180,E1 -7010.45,E2 -7010.45} C_VEL
LIN {X 0,Y 481.837,Z 411.264,A -85,B 0,C 180,E1 -7011.187,E2 -7011.187} C_VEL
LIN {X 0,Y 481.577,Z 418.601,A -85,B 0,C 180,E1 -7012.027,E2 -7012.027} C_VEL
LIN {X 0,Y 481.353,Z 426.415,A -85,B 0,C 180,E1 -7013.142,E2 -7013.142} C_VEL
LIN {X 0,Y 481.225,Z 431.824,A -85,B 0,C 180,E1 -7014.128,E2 -7014.128} C_VEL
LIN {X 0,Y 480.994,Z 435.629,A -85,B 0,C 180,E1 -7014.967,E2 -7014.967} C_VEL
LIN {X 0,Y 481.08,Z 438.693,A -85,B 0,C 180,E1 -7015.807,E2 -7015.807} C_VEL
LIN {X 0,Y 480.979,Z 441.089,A -85,B 0,C 180,E1 -7016.645,E2 -7016.645} C_VEL
LIN {X 0,Y 480.916,Z 442.923,A -85,B 0,C 180,E1 -7017.483,E2 -7017.483} C_VEL
LIN {X 0,Y 480.828,Z 444.241,A -85,B 0,C 180,E1 -7018.321,E2 -7018.321} C_VEL
LIN {X 0,Y 480.764,Z 445.066,A -85,B 0,C 180,E1 -7019.158,E2 -7019.158} C_VEL
LIN {X 0,Y 480.75,Z 445.36,A -85,B 0,C 180,E1 -7019.996,E2 -7019.996} C_VEL
LIN {X 0,Y 480.764,Z 445.057,A -85,B 0,C 180,E1 -7020.833,E2 -7020.833} C_VEL
LIN {X 0,Y 480.826,Z 444.261,A -85,B 0,C 180,E1 -7021.671,E2 -7021.671} C_VEL
LIN {X 0,Y 480.888,Z 442.973,A -85,B 0,C 180,E1 -7022.509,E2 -7022.509} C_VEL
LIN {X 0,Y 481.002,Z 439.988,A -85,B 0,C 180,E1 -7023.766,E2 -7023.766} C_VEL
LIN {X 0,Y 481.02,Z 437.267,A -85,B 0,C 180,E1 -7024.605,E2 -7024.605} C_VEL
LIN {X 0,Y 481.059,Z 433.906,A -85,B 0,C 180,E1 -7025.445,E2 -7025.445} C_VEL
LIN {X 0,Y 481.392,Z 428.508,A -85,B 0,C 180,E1 -7026.513,E2 -7026.513} C_VEL
LIN {X 0,Y 481.382,Z 423.6,A -85,B 0,C 180,E1 -7027.314,E2 -7027.314} C_VEL
LIN {X 0,Y 481.559,Z 417.21,A -85,B 0,C 180,E1 -7028.176,E2 -7028.176} C_VEL
LIN {X 0,Y 481.775,Z 410.645,A -85,B 0,C 180,E1 -7028.912,E2 -7028.912} C_VEL
LIN {X 0,Y 482.011,Z 402.699,A -85,B 0,C 180,E1 -7029.648,E2 -7029.648} C_VEL
LIN {X 0,Y 482.302,Z 392.801,A -85,B 0,C 180,E1 -7030.384,E2 -7030.384} C_VEL
LIN {X 0,Y 482.542,Z 381.216,A -85,B 0,C 180,E1 -7031.016,E2 -7031.016} C_VEL
LIN {X 0,Y 482.683,Z 371.909,A -85,B 0,C 180,E1 -7031.384,E2 -7031.384} C_VEL
LIN {X 0,Y 482.815,Z 362.257,A -85,B 0,C 180,E1 -7031.647,E2 -7031.647} C_VEL
LIN {X 0,Y 483.147,Z 296.568,A -85,B 0,C 180,E1 -7032.745,E2 -7032.745} C_VEL
LIN {X 0,Y 481.555,Z 286.664,A -85,B 0,C 180,E1 -7032.965,E2 -7032.965} C_VEL
LIN {X 0,Y 481.793,Z 273.921,A -85,B 0,C 180,E1 -7036.085,E2 -7036.085} C_VEL
LIN {X 0,Y 481.907,Z 266.955,A -85,B 0,C 180,E1 -7037.828,E2 -7037.828} C_VEL
LIN {X 0,Y 481.774,Z 265.287,A -85,B 0,C 180,E1 -7038.287,E2 -7038.287} C_VEL
LIN {X 0,Y 481.632,Z 265.305,A -85,B 0,C 180,E1 -7041.39,E2 -7041.39} C_VEL
LIN {X 0,Y 481.632,Z 265.301,A -85,B 0,C 180,E1 -7044.109,E2 -7044.109} C_VEL
LIN {X 0,Y 481.635,Z 265.304,A -85,B 0,C 180,E1 -7047.112,E2 -7047.112} C_VEL
LIN {X 0,Y 481.644,Z 265.302,A -85,B 0,C 180,E1 -7049.737,E2 -7049.737} C_VEL
LIN {X 0,Y 481.648,Z 265.3,A -85,B 0,C 180,E1 -7052.669,E2 -7052.669} C_VEL
LIN {X 0,Y 481.606,Z 265.308,A -85,B 0,C 180,E1 -7055.705,E2 -7055.705} C_VEL
LIN {X 0,Y 481.639,Z 265.301,A -85,B 0,C 180,E1 -7058.854,E2 -7058.854} C_VEL
LIN {X 0,Y 481.614,Z 265.307,A -85,B 0,C 180,E1 -7061.906,E2 -7061.906} C_VEL
LIN {X 0,Y 481.62,Z 265.302,A -85,B 0,C 180,E1 -7064.453,E2 -7064.453} C_VEL
LIN {X 0,Y 481.611,Z 265.307,A -85,B 0,C 180,E1 -7067.834,E2 -7067.834} C_VEL
LIN {X 0,Y 481.621,Z 265.302,A -85,B 0,C 180,E1 -7070.649,E2 -7070.649} C_VEL
LIN {X 0,Y 481.588,Z 265.308,A -85,B 0,C 180,E1 -7073.371,E2 -7073.371} C_VEL
LIN {X 0,Y 481.645,Z 265.3,A -85,B 0,C 180,E1 -7075.268,E2 -7075.268} C_VEL
LIN {X 0,Y 481.013,Z 265.382,A -85,B 0,C 180,E1 -7075.966,E2 -7075.966} C_VEL
LIN {X 0,Y 478.137,Z 265.741,A -85,B 0,C 180,E1 -7077.1,E2 -7077.1} C_VEL
LIN {X 0,Y 475.683,Z 266.045,A -85,B 0,C 180,E1 -7078.013,E2 -7078.013} C_VEL
LIN {X 0,Y 474.634,Z 266.174,A -85,B 0,C 180,E1 -7078.72,E2 -7078.72} C_VEL
LIN {X 0,Y 474.553,Z 266.183,A -85,B 0,C 180,E1 -7078.959,E2 -7078.959} C_VEL
LIN {X 0,Y 474.599,Z 266.18,A -85,B 0,C 180,E1 -7081.713,E2 -7081.713} C_VEL
LIN {X 0,Y 474.62,Z 266.178,A -85,B 0,C 180,E1 -7084.574,E2 -7084.574} C_VEL
LIN {X 0,Y 474.548,Z 266.183,A -85,B 0,C 180,E1 -7087.352,E2 -7087.352} C_VEL
LIN {X 0,Y 474.601,Z 266.181,A -85,B 0,C 180,E1 -7090.086,E2 -7090.086} C_VEL
LIN {X 0,Y 474.595,Z 266.181,A -85,B 0,C 180,E1 -7092.771,E2 -7092.771} C_VEL
LIN {X 0,Y 474.592,Z 266.178,A -85,B 0,C 180,E1 -7095.418,E2 -7095.418} C_VEL
LIN {X 0,Y 474.683,Z 266.169,A -85,B 0,C 180,E1 -7098.036,E2 -7098.036} C_VEL
LIN {X 0,Y 474.672,Z 266.168,A -85,B 0,C 180,E1 -7101.484,E2 -7101.484} C_VEL
LIN {X 0,Y 474.731,Z 266.161,A -85,B 0,C 180,E1 -7104.05,E2 -7104.05} C_VEL
LIN {X 0,Y 474.842,Z 266.148,A -85,B 0,C 180,E1 -7107.454,E2 -7107.454} C_VEL
LIN {X 0,Y 474.848,Z 266.146,A -85,B 0,C 180,E1 -7109.999,E2 -7109.999} C_VEL
LIN {X 0,Y 474.841,Z 266.15,A -85,B 0,C 180,E1 -7112.543,E2 -7112.543} C_VEL
LIN {X 0,Y 474.729,Z 266.161,A -85,B 0,C 180,E1 -7115.947,E2 -7115.947} C_VEL
LIN {X 0,Y 474.674,Z 266.169,A -85,B 0,C 180,E1 -7118.513,E2 -7118.513} C_VEL
LIN {X 0,Y 474.679,Z 266.168,A -85,B 0,C 180,E1 -7121.961,E2 -7121.961} C_VEL
LIN {X 0,Y 474.618,Z 266.177,A -85,B 0,C 180,E1 -7125.768,E2 -7125.768} C_VEL
LIN {X 0,Y 474.604,Z 266.18,A -85,B 0,C 180,E1 -7129.011,E2 -7129.011} C_VEL
LIN {X 0,Y 474.534,Z 266.188,A -85,B 0,C 180,E1 -7131.73,E2 -7131.73} C_VEL
LIN {X 0,Y 474.603,Z 266.176,A -85,B 0,C 180,E1 -7134.494,E2 -7134.494} C_VEL
LIN {X 0,Y 474.64,Z 266.177,A -85,B 0,C 180,E1 -7137.34,E2 -7137.34} C_VEL
LIN {X 0,Y 474.552,Z 266.183,A -85,B 0,C 180,E1 -7140.813,E2 -7140.813} C_VEL
LIN {X 0,Y 474.582,Z 266.182,A -85,B 0,C 180,E1 -7143.986,E2 -7143.986} C_VEL
LIN {X 0,Y 474.521,Z 266.187,A -85,B 0,C 180,E1 -7146.902,E2 -7146.902} C_VEL
LIN {X 0,Y 474.617,Z 266.179,A -85,B 0,C 180,E1 -7149.657,E2 -7149.657} C_VEL
LIN {X 0,Y 474.601,Z 266.177,A -85,B 0,C 180,E1 -7152.933,E2 -7152.933} C_VEL
LIN {X 0,Y 474.569,Z 266.185,A -85,B 0,C 180,E1 -7155.899,E2 -7155.899} C_VEL
LIN {X 0,Y 474.598,Z 266.177,A -85,B 0,C 180,E1 -7159.042,E2 -7159.042} C_VEL
LIN {X 0,Y 474.571,Z 266.182,A -85,B 0,C 180,E1 -7161.707,E2 -7161.707} C_VEL
LIN {X 0,Y 474.587,Z 266.182,A -85,B 0,C 180,E1 -7164.73,E2 -7164.73} C_VEL
LIN {X 0,Y 474.595,Z 266.178,A -85,B 0,C 180,E1 -7167.792,E2 -7167.792} C_VEL
LIN {X 0,Y 474.583,Z 266.182,A -85,B 0,C 180,E1 -7170.889,E2 -7170.889} C_VEL
LIN {X 0,Y 474.591,Z 266.178,A -85,B 0,C 180,E1 -7173.631,E2 -7173.631} C_VEL
LIN {X 0,Y 474.599,Z 266.18,A -85,B 0,C 180,E1 -7176.646,E2 -7176.646} C_VEL
LIN {X 0,Y 474.62,Z 266.175,A -85,B 0,C 180,E1 -7180.094,E2 -7180.094} C_VEL
LIN {X 0,Y 474.606,Z 266.18,A -85,B 0,C 180,E1 -7182.778,E2 -7182.778} C_VEL
LIN {X 0,Y 474.616,Z 266.177,A -85,B 0,C 180,E1 -7185.425,E2 -7185.425} C_VEL
LIN {X 0,Y 474.678,Z 266.167,A -85,B 0,C 180,E1 -7188.042,E2 -7188.042} C_VEL
LIN {X 0,Y 474.686,Z 266.169,A -85,B 0,C 180,E1 -7191.491,E2 -7191.491} C_VEL
LIN {X 0,Y 474.739,Z 266.159,A -85,B 0,C 180,E1 -7194.057,E2 -7194.057} C_VEL
LIN {X 0,Y 474.86,Z 266.147,A -85,B 0,C 180,E1 -7197.46,E2 -7197.46} C_VEL
LIN {X 0,Y 474.862,Z 266.145,A -85,B 0,C 180,E1 -7200.004,E2 -7200.004} C_VEL
LIN {X 0,Y 474.865,Z 266.144,A -85,B 0,C 180,E1 -7202.549,E2 -7202.549} C_VEL
LIN {X 0,Y 474.733,Z 266.163,A -85,B 0,C 180,E1 -7205.952,E2 -7205.952} C_VEL
LIN {X 0,Y 474.694,Z 266.165,A -85,B 0,C 180,E1 -7208.518,E2 -7208.518} C_VEL
LIN {X 0,Y 474.692,Z 266.168,A -85,B 0,C 180,E1 -7211.966,E2 -7211.966} C_VEL
LIN {X 0,Y 474.678,Z 266.172,A -85,B 0,C 180,E1 -7215.46,E2 -7215.46} C_VEL
LIN {X 0,Y 474.65,Z 266.171,A -85,B 0,C 180,E1 -7219.014,E2 -7219.014} C_VEL
LIN {X 0,Y 474.579,Z 266.184,A -85,B 0,C 180,E1 -7221.733,E2 -7221.733} C_VEL
LIN {X 0,Y 474.619,Z 266.177,A -85,B 0,C 180,E1 -7224.498,E2 -7224.498} C_VEL
LIN {X 0,Y 474.631,Z 266.173,A -85,B 0,C 180,E1 -7227.327,E2 -7227.327} C_VEL
LIN {X 0,Y 474.596,Z 266.18,A -85,B 0,C 180,E1 -7230.234,E2 -7230.234} C_VEL
LIN {X 0,Y 474.61,Z 266.175,A -85,B 0,C 180,E1 -7233.226,E2 -7233.226} C_VEL
LIN {X 0,Y 474.574,Z 266.183,A -85,B 0,C 180,E1 -7236.328,E2 -7236.328} C_VEL
LIN {X 0,Y 474.597,Z 266.178,A -85,B 0,C 180,E1 -7239.646,E2 -7239.646} C_VEL
LIN {X 0,Y 474.571,Z 266.183,A -85,B 0,C 180,E1 -7242.942,E2 -7242.942} C_VEL
LIN {X 0,Y 474.578,Z 266.18,A -85,B 0,C 180,E1 -7245.894,E2 -7245.894} C_VEL
LIN {X 0,Y 474.598,Z 266.18,A -85,B 0,C 180,E1 -7249.048,E2 -7249.048} C_VEL
LIN {X 0,Y 474.598,Z 266.177,A -85,B 0,C 180,E1 -7251.709,E2 -7251.709} C_VEL
LIN {X 0,Y 474.617,Z 266.178,A -85,B 0,C 180,E1 -7254.727,E2 -7254.727} C_VEL
LIN {X 0,Y 474.625,Z 266.174,A -85,B 0,C 180,E1 -7257.789,E2 -7257.789} C_VEL
LIN {X 0,Y 474.595,Z 266.181,A -85,B 0,C 180,E1 -7260.894,E2 -7260.894} C_VEL
LIN {X 0,Y 474.581,Z 266.181,A -85,B 0,C 180,E1 -7263.626,E2 -7263.626} C_VEL
LIN {X 0,Y 474.679,Z 266.374,A -85,B 0,C 180,E1 -7266.033,E2 -7266.033} C_VEL
LIN {X 0,Y 475.999,Z 275.125,A -85,B 0,C 180,E1 -7267.885,E2 -7267.885} C_VEL
LIN {X 0,Y 475.437,Z 290.775,A -85,B 0,C 180,E1 -7271.024,E2 -7271.024} C_VEL
LIN {X 0,Y 474.851,Z 307.304,A -85,B 0,C 180,E1 -7274.29,E2 -7274.29} C_VEL
LIN {X 0,Y 474.517,Z 320.505,A -85,B 0,C 180,E1 -7276.872,E2 -7276.872} C_VEL
LIN {X 0,Y 476.284,Z 336.002,A -85,B 0,C 180,E1 -7277.19,E2 -7277.19} C_VEL
LIN {X 0,Y 475.743,Z 398.384,A -85,B 0,C 180,E1 -7278.255,E2 -7278.255} C_VEL
LIN {X 0,Y 475.5,Z 410.06,A -85,B 0,C 180,E1 -7278.6,E2 -7278.6} C_VEL
LIN {X 0,Y 475.222,Z 421.47,A -85,B 0,C 180,E1 -7279.133,E2 -7279.133} C_VEL
